//disrupt calling SystemFlowControl via MAIN() when mode is switched and call SwitchMode()
IF ((SwitchToLoading.Q OR SwitchToUnloading.Q) OR NOT bFinishedSwitchMode) AND bSetStatusOn THEN
	SwitchMode(bSwitchToLoading := bLoading,
		bFinishedSwitchMode => bFinishedSwitchMode);
END_IF;

//pumps
PU305.GetState_Profibus();
PU305(bSetStatusOnAutomatic := bSetStatusOn_PU305,
	fSetPointAutomatic := fSetPoint,
	bAlgorithmPermission := bAlgorithmPermission,
	nControlModeAutomatic := 0);
PU305.SetState_Profibus();

PU306.GetState_Profibus();
PU306(bSetStatusOnAutomatic := bSetStatusOn_PU306,
	fSetPointAutomatic := fSetPoint,
	bAlgorithmPermission := bAlgorithmPermission,
	nControlModeAutomatic := 0);
PU306.SetState_Profibus();

//valves
SV305.GetState_AI();
SV305(bSetStatusOnAutomatic := bSetStatusOn_SV305,
	fSetPointAutomatic := fSetPoint_SV305,
	bAlgorithmPermission := bAlgorithmPermission,
	nControlModeAutomatic := 0);
SV305.SetState_AO();

SV306.GetState_AI();
SV306(bSetStatusOnAutomatic := bSetStatusOn_SV306,
	fSetPointAutomatic := fSetPoint_SV306,
	bAlgorithmPermission := bAlgorithmPermission,
	nControlModeAutomatic := 0);
SV306.SetState_AO();

WMZ305(aHeatCounterTelegramm := aTelegramm_WMZ305);

IF bLoading THEN
	localState.fHeatFlowRate := -PU305.fVolumeFlowRate/3.6*4.2*(WMZ305.fFeedTemperature-WMZ305.fReturnTemperature);
	nControlMode_SV307 := 2; //cooling
ELSE
	localState.fHeatFlowRate := PU306.fVolumeFlowRate/3.6*4.2*(WMZ305.fFeedTemperature-WMZ305.fReturnTemperature);
	nControlMode_SV307 := 1; //heating
END_IF

SV307.GetState_AI();
SV307(bSetStatusOnAutomatic := bSetStatusOn_SV307,
	fSetPointAutomatic := fTemperatureBufferStorageSetPoint,
	bAlgorithmPermission := bAlgorithmPermission,
	fTemperatureExternal := fTemperatureBufferStorage,
	fThermalPowerExternal := localState.fHeatFlowRate,
	nControlModeAutomatic := nControlMode_SV307);
SV307.SetState_AO();

METHOD PROTECTED  CheckError : BOOL
VAR_INPUT
END_VAR
VAR_OUTPUT
	bError : BOOL;
END_VAR
VAR
	bError_PUx05 : BOOL;
END_VAR
//check for pump error
bError_PUx05 := PU305.bError OR PU306.bError;
END_METHOD

METHOD PROTECTED  Operational : BOOL
VAR_INPUT
END_VAR
VAR_OUTPUT
	bSwitchToWorking : BOOL := FALSE;
END_VAR
IF PU305.bStatusOn OR PU306.bStatusOn THEN
	bSwitchToWorking := TRUE;
END_IF
END_METHOD

METHOD PROTECTED  RampDown : BOOL
VAR_INPUT
END_VAR
VAR_OUTPUT
	bRampDownFinished : BOOL := FALSE;
END_VAR
bSetStatusOn_PU305 := FALSE;
bSetStatusOn_PU306 := FALSE;

IF NOT PU305.bStatusOn AND NOT PU306.bStatusOn THEN
	bSetStatusOn_SV305 := FALSE;
	bSetStatusOn_SV306 := FALSE;
	bSetStatusOn_SV307 := FALSE;
	IF SV305.fOperatingPoint<20 AND SV306.fOperatingPoint<20 AND SV307.fOperatingPoint<20 THEN
		bRampDownFinished := TRUE;
	END_IF
END_IF
END_METHOD

METHOD PROTECTED  RampUp : BOOL
VAR_INPUT
END_VAR
VAR_OUTPUT
	bRampUpFinished : BOOL := FALSE;
END_VAR
bSetStatusOn_SV305 := TRUE;
bSetStatusOn_SV306 := TRUE;
bSetStatusOn_SV307 := TRUE;

//SV307 should not be checked in ramp up to prevent chattering when sv control thermal power
IF bLoading THEN
	fSetPoint_SV305 := 100;
	fSetPoint_SV306 := 0;
	IF SV305.fOperatingPoint>80 AND SV306.fOperatingPoint<20 THEN
		bSetStatusOn_PU305 := TRUE;	
		bSetStatusOn_PU306 := FALSE;	
		bRampUpFinished := TRUE;	
	END_IF
ELSE
	fSetPoint_SV305 := 0;
	fSetPoint_SV306 := 100;
	IF SV305.fOperatingPoint<20 AND SV306.fOperatingPoint>80 THEN
		bSetStatusOn_PU305 := FALSE;	
		bSetStatusOn_PU306 := TRUE;		
		bRampUpFinished := TRUE;
	END_IF
END_IF
END_METHOD

METHOD PRIVATE SelectLocalControlMode : BOOL
VAR_INPUT
END_VAR
IF control.bManualModeActivated THEN
	bLoading := localSetParameters.bLoadingManual;
ELSIF control.bAlgorithmModeActivated AND bAlgorithmPermission THEN
	bLoading := localSetParameters.bLoadingAlgorithm;
ELSE
	bLoading := bLoadingAutomatic;
END_IF
END_METHOD

METHOD PROTECTED   SetSetPointLimits : BOOL
VAR_INPUT
END_VAR
aSetPointLimits[1] := localDefaultParameters.aSetPointLimitsTemperature[1];
aSetPointLimits[2] := localDefaultParameters.aSetPointLimitsTemperature[2];
END_METHOD

METHOD PROTECTED  SetState : BOOL
VAR_INPUT
END_VAR
VAR_OUTPUT
END_VAR
IF bLoading THEN
	fOperatingPoint := PU305.fOperatingPoint;
ELSE
	fOperatingPoint := PU306.fOperatingPoint;
END_IF

IF PU305.bStatusOn THEN
	localState.bLoading := TRUE;
ELSE
	localState.bLoading := FALSE;		
END_IF

controlState.bStatusOn := bSetStatusOn;
setPointState.aSetPointLimits := aSetPointLimits;
setPointState.fSetPoint := fSetPoint;
setPointState.fOperatingPoint := fOperatingPoint;
setPointState.sSetPointUnit := 'percent';
setPointState.sOperatingPointUnit := 'percent';
END_METHOD

PROPERTY ST_DefaultParameters : REFERENCE TO ST_VSIStorageSystemDefaultParameters
SET
localDefaultParameters := ST_DefaultParameters;
END_SET
END_PROPERTY

METHOD PRIVATE SwitchMode : BOOL
VAR_INPUT
	bSwitchToLoading : BOOL; //if false switch to cooling
END_VAR
VAR_OUTPUT
	bFinishedSwitchMode : BOOL := FALSE;
END_VAR
VAR_INST
	bRampDownFinished : BOOL := FALSE;
END_VAR
//check system state
IF bRampDownFinished THEN
	IF bSwitchToLoading THEN
		fSetPoint_SV305 := 100;
		fSetPoint_SV306 := 0;
		IF SV305.fOperatingPoint>80 AND SV306.fOperatingPoint<20 THEN
			//reset instant variable and switch on pump
			bRampDownFinished := FALSE;			
			bFinishedSwitchMode := TRUE;
			bSetStatusOn_PU305 := TRUE;
		END_IF
		
	ELSE
		fSetPoint_SV305 := 0;
		fSetPoint_SV306 := 100;
		IF SV305.fOperatingPoint<20 AND SV306.fOperatingPoint>80 THEN
			//reset instant variable and switch on pump
			bRampDownFinished := FALSE;			
			bFinishedSwitchMode := TRUE;
			bSetStatusOn_PU306 := TRUE;
		END_IF
	END_IF
ELSE
	bSetStatusOn_PU305 := FALSE;
	bSetStatusOn_PU306 := FALSE;
	IF NOT PU305.bStatusOn AND NOT PU306.bStatusOn THEN
		bRampDownFinished := TRUE;
	END_IF
END_IF
END_METHOD

METHOD PROTECTED  Working : BOOL
VAR_INPUT
END_VAR
VAR_OUTPUT
	bSwitchToOperational : BOOL := FALSE;
END_VAR
//empty method
END_METHOD

END_FUNCTION_BLOCK

// ---- POUs/03 Storages/FB_VSIStorage.TcPOU
FUNCTION_BLOCK FB_VSIStorage
VAR_INPUT
END_VAR
VAR_OUTPUT
	{attribute 'OPC.UA.DA' := '1'}	
	localState : ST_VSIStorageState;
END_VAR
VAR
	UpperTemperatureSensor : FB_TemperatureSensor; //upper temperature sensor
	MidTemperatureSensor : FB_TemperatureSensor; //mid temperature sensor
	LowerTemperatureSensor : FB_TemperatureSensor; //lower temperature sensor
END_VAR

//sensors
UpperTemperatureSensor();
MidTemperatureSensor();
LowerTemperatureSensor();

//get sensor inputs
UpperTemperatureSensor.GetState_AI();
MidTemperatureSensor.GetState_AI();
LowerTemperatureSensor.GetState_AI();

//set outputs
localState.fUpperTemperature := UpperTemperatureSensor.fTemperature;
localState.fMidTemperature := MidTemperatureSensor.fTemperature;
localState.fLowerTemperature := LowerTemperatureSensor.fTemperature;

END_FUNCTION_BLOCK

// ---- POUs/01 Actuators/ConsumerUnits/FB_MAFAC_Java.TcPOU
FUNCTION_BLOCK FB_MAFAC_Java
VAR_INPUT
END_VAR
VAR_OUTPUT
	bStatusOn : BOOL;
	bError_Connection : BOOL;
END_VAR
VAR
	OPC_UA				: FB_OPC_UA_READ;
	stOPC_UA_Server		: ST_OPC_UA_Server;
	sOPC_UA_Server_URL 	: STRING;
	sNamespaceName		: STRING;
	aNodes				: ARRAY[1..1] OF ST_OPC_UANode;
	nNodeCount			: UDINT := 1;
	stIndexRange		: ARRAY [1..nMaxIndexRange] OF ST_UAIndexRange;
	currentNode			: UDINT := 1;
	
	bStatusOn_CoolingLubricant : BOOL;
	bStatusOn_Machine : BOOL;
	
	// timer
	bStartTimer : BOOL;
	Timer : TON;
END_VAR

sOPC_UA_Server_URL 	:= GlobalVariables.sIP_MAFAC_Java;
sNamespaceName 		:= 'http://www.boschrexroth.com/IndraLogic';

(*Define Nodes to Read*)
aNodes[1].NodeID.sIdentifier			:= 'Application.UserVarGlobal.Beheizung_rot_Aktiv';
aNodes[1].NodeID.eIdentifierType		:= eUAIdentifierType_String;
aNodes[1].SizeOfDataType				:= SIZEOF(eUAType_Boolean);
aNodes[1].NodeAddInfo.nIndexRangeCount 	:= 0;
aNodes[1].NodeAddInfo.stIndexRange		:= stIndexRange;
aNodes[1].TargetVar						:= ADR(bStatusOn);
bError_Connection := OPC_UA.bError_Connection;
Timer(IN := bStartTimer,
	PT := T#5S);

bStartTimer := TRUE;
IF Timer.Q THEN
	OPC_UA(
		stNode				:= aNodes[currentNode],
		sOPC_UA_Server_Url 	:= sOPC_UA_Server_URL,
		sNamespaceName		:= sNamespaceName);
	currentNode := currentNode + 1;
	IF currentNode > nNodeCount THEN
		currentNode := 1;
	END_IF
	bStartTimer := FALSE;
END_IF

END_FUNCTION_BLOCK

// ---- POUs/01 Actuators/ConsumerUnits/FB_BvL_CleaningSystem.TcPOU
FUNCTION_BLOCK FB_BvL_CleaningSystem
VAR_INPUT
END_VAR
VAR_OUTPUT
	bError_Connection : BOOL;
	bHNHT_Demand : BOOL; 
END_VAR
VAR
	//I/O-Links
	Technical_Heat_RZ_SV AT %I* : BOOL;
	Technical_Heat_RZ_PWW AT %I* : BOOL;
	Technical_Heat_RZ_UWP AT %I* : BOOL;
	Technical_Heat_SZ_SV AT %I* : BOOL;
	Technical_Heat_SZ_PWW AT %I* : BOOL;
	Technical_Heat_SZ_UWP AT %I* : BOOL; 
	ConnectionStatus_OPC_BvL AT %I* : BOOL;
END_VAR

bHNHT_Demand := (Technical_Heat_RZ_PWW OR Technical_Heat_RZ_SV OR Technical_Heat_RZ_UWP OR Technical_Heat_SZ_PWW OR Technical_Heat_SZ_SV OR Technical_Heat_SZ_UWP) AND ConnectionStatus_OPC_BvL;
bError_Connection := NOT ConnectionStatus_OPC_BvL;

END_FUNCTION_BLOCK

// ---- POUs/05 Thermal Networks/FB_Ambient.TcPOU
FUNCTION_BLOCK FB_Ambient
VAR_INPUT
	sIPAddress : STRING(15);
END_VAR
VAR_OUTPUT
	{attribute 'OPC.UA.DA' := '1'}
	localState : ST_AmbientState;
END_VAR
VAR
	WeatherStation : FB_WeatherStation;
	AmbientTemperatureSensor_Container : FB_TemperatureSensor_KL3214;
	HallTemperatureSensor_Section1 : FB_TemperatureSensor;
	HallTemperatureSensor_Section2 : FB_TemperatureSensor;
	HallTemperatureSensor_Section3 : FB_TemperatureSensor;
	RoomTemperatureSensor_Container : FB_TemperatureSensor;
	
	//modbus tcp communication
	ModbusReader_250 : FB_MBReadRegs; //read regs from 250 on
	
	//define array to store data from every ModbusReader
	aModbus_250 : ARRAY [0..31] OF WORD;
	
	//modbus timer
	bReadModbus	: BOOL := FALSE;
	bWriteModbus_SeminarRoom : BOOL := FALSE; 
	bStartTimer : BOOL;
	TimerReader : TON; 
END_VAR

WeatherStation();
HallTemperatureSensor_Section1();
HallTemperatureSensor_Section1.GetState_AI();
HallTemperatureSensor_Section2();
HallTemperatureSensor_Section2.GetState_AI();
HallTemperatureSensor_Section3();
HallTemperatureSensor_Section3.GetState_AI();
AmbientTemperatureSensor_Container();
AmbientTemperatureSensor_Container.GetState_AI();
RoomTemperatureSensor_Container();
RoomTemperatureSensor_Container.GetState_AI();


//add ambient temperature rain etc. from weather station
localState.fOutsideTemperature_Container := AmbientTemperatureSensor_Container.fTemperature;
localState.fOutsideTemperature := WeatherStation.fTemperature;
localState.fOutsideTemperature_Mean := WeatherStation.fMeanTemperature;
localState.bRain := WeatherStation.bRain;
localState.fDawn := WeatherStation.fDawn;
localState.fWindSpeed := WeatherStation.fWindSpeed;
localState.fHallTemperature := HallTemperatureSensor_Section2.fTemperature;
localState.fRoomTemperature_Container := RoomTemperatureSensor_Container.fTemperature;


//Start and check timer for 2s interval
TimerReader(IN := bStartTimer,
	PT := T#2S);
	
bStartTimer := TRUE;
IF TimerReader.Q THEN
	bReadModbus := TRUE;
	bStartTimer := FALSE;	
END_IF
	

ModbusReader_250(
	sIPAddr := sIPAddress,
	nTCPPort := 502,
	nUnitID := 255,
	nQuantity := 30,
	nMBAddr := 250,
	cbLength := 60,
	pDestAddr := ADR(aModbus_250),
	bExecute := bReadModbus,
	tTimeout  := T#20S);
	
bReadModbus := FALSE;

//seminar room
localState.fTemperatureSeminarRoom := INT_TO_REAL(WORD_TO_INT(aModbus_250[19]))/10; 
localState.fCO2SeminarRoom := INT_TO_REAL(WORD_TO_INT(aModbus_250[17])); 
//student room
localState.fTemperatureStudentRoom := INT_TO_REAL(WORD_TO_INT(aModbus_250[28])); 
localState.fCO2StudentRoom := INT_TO_REAL(WORD_TO_INT(aModbus_250[27]));

METHOD GetState : BOOL
VAR_INPUT
END_VAR
//seminar room
localState.fTemperatureSeminarRoom := INT_TO_REAL(WORD_TO_INT(aModbus_250[19]))/10; 
localState.fCO2SeminarRoom := INT_TO_REAL(WORD_TO_INT(aModbus_250[17])); 

//student room
localState.fTemperatureStudentRoom := INT_TO_REAL(WORD_TO_INT(aModbus_250[28])); 
localState.fCO2StudentRoom := INT_TO_REAL(WORD_TO_INT(aModbus_250[27]));
END_METHOD

END_FUNCTION_BLOCK

// ---- POUs/02 Sensors/FB_WeatherStation.TcPOU
FUNCTION_BLOCK FB_WeatherStation
VAR_INPUT
END_VAR
VAR_OUTPUT
	fWindSpeed 		: REAL;
	fTemperature	: REAL;
	fMeanTemperature : REAL;
	fDawn 			: REAL;
	bRain 			: BOOL;
END_VAR
VAR
	bInit_done : BOOL := FALSE;
	
	// communication with KL6301 terminal
	KL6301_Terminal			: KL6301;
	KL6301_Error_Trigger	: r_Trig;
	KL6301_group_0_0_1		: EIB_GROUP_ADDR := (MAIN:=0, SUB_MAIN:=0, NUMBER:=1);
	KL6301_IN 				AT %I* : ARRAY[1..24]OF BYTE;
	KL6301_OUT 				AT %Q* : ARRAY[1..24]OF BYTE;
	
	Group_0_0_1		: EIB_GROUP_ADDR := (MAIN:=0,SUB_MAIN:=0,NUMBER:=1);
	Group_0_0_2		: EIB_GROUP_ADDR := (MAIN:=0,SUB_MAIN:=0,NUMBER:=2);
	Group_0_0_3		: EIB_GROUP_ADDR := (MAIN:=0,SUB_MAIN:=0,NUMBER:=3);
	Group_0_0_4		: EIB_GROUP_ADDR := (MAIN:=0,SUB_MAIN:=0,NUMBER:=4);

	recWindSpeed	: EIB_2OCTET_FLOAT_REC;
	recTemperature	: EIB_2OCTET_FLOAT_REC;
	recDawn			: EIB_2OCTET_FLOAT_REC;
	recRain			: EIB_BIT_REC;
	
	//clock
	stDefaultParameters_Clock : ST_ClockDefaultParameters := (tTaskCycleTime := GlobalVariables.tCtrlCycleTime_MAIN, tCtrlCycleTime := T#1M);
	Clock : FB_Clock := (ST_DefaultParameters := stDefaultParameters_Clock);
	Moving_Average_Temperature : FB_CTRL_MOVING_AVERAGE;
	bInit_Average_Temperature : BOOL;
END_VAR

//initialize clock
Clock();

//read and write to terminal
KL6301_Terminal(KL6301_IN:=KL6301_IN, KL6301_OUT:=KL6301_OUT);
KL6301_Error_Trigger(CLK := KL6301_Terminal.bError);

//initialize terminal
IF (NOT bInit_done) THEN
	bInit_done := InitializeTerminal();
END_IF

IF(KL6301_Terminal.bReady) THEN
	recWindSpeed(
		Group_Address := Group_0_0_1,
		strData_Rec := KL6301_Terminal.str_Data_Rec
	);

	recTemperature(
		Group_Address := Group_0_0_2,
		strData_Rec := KL6301_Terminal.str_Data_Rec
	);

	recDawn(
		Group_Address := Group_0_0_3,
		strData_Rec := KL6301_Terminal.str_Data_Rec
	);

	recRain(
		Group_Address := Group_0_0_4,
		strData_Rec := KL6301_Terminal.str_Data_Rec
	);

	fWindSpeed := recWindSpeed.rData;
	fTemperature := recTemperature.rData;
	fDawn := recDawn.rData;
	bRain := recRain.bData;
END_IF

//calculate moving average temperatrue
CalculateAverageTemperature(fActualTemperature := fTemperature, fMeanTemperature => fMeanTemperature);

METHOD CalculateAverageTemperature : REAL
VAR_INPUT
	fActualTemperature : REAL;
END_VAR
VAR_OUTPUT
	fMeanTemperature : REAL;
END_VAR
VAR_INST
	fTemperature_init : REAL;
	fHours_Moving_Average : UINT := 6;
	fMeanTemperature_Summer_init : REAL := 22;
	fMeanTemperature_Winter_init : REAL := 5;
	
	stParameters_Average_Temperature : ST_CTRL_MOVING_AVERAGE_PARAMS;
	aTemperatureBuffer 				: ARRAY [1..360] OF FLOAT := [360(15)];
END_VAR
//calculate initialization temperature
IF Clock.stClockState.sintMonth>4 AND Clock.stClockState.sintMonth<10 THEN
	//summer
	fTemperature_init := fMeanTemperature_Summer_init;
ELSE
	//winter	
	fTemperature_init := fMeanTemperature_Winter_init;
END_IF

stParameters_Average_Temperature.tCtrlCycleTime := T#60S;
stParameters_Average_Temperature.tTaskCycleTime := GlobalVariables.tTaskCycleTime_MAIN;
stParameters_Average_Temperature.nSamplesToFilter := fHours_Moving_Average*60; (* 1min= 60 sec*)
stParameters_Average_Temperature.pWorkArray_ADR := ADR(aTemperatureBuffer);
stParameters_Average_Temperature.nWorkArray_SIZEOF := SIZEOF(aTemperatureBuffer);

Moving_Average_Temperature(
	fIn := fActualTemperature,
	fManSyncValue := 15,
	bSync := FALSE,
	eMode := 2,
	bHold := FALSE,
	stParams := stParameters_Average_Temperature);
fMeanTemperature := LREAL_TO_REAL(Moving_Average_Temperature.fOut);
END_METHOD

METHOD InitializeTerminal : BOOL
VAR_INPUT
END_VAR
VAR_OUTPUT
	bInit_done : BOOL := FALSE;
END_VAR
KL6301_Terminal.EIB_PHYS_ADDR.Area:=1;
KL6301_Terminal.EIB_PHYS_ADDR.Line:=1;
KL6301_Terminal.EIB_PHYS_ADDR.Device:=5;
KL6301_Terminal.EIB_GROUP_FILTER[1].GROUP_ADDR:=KL6301_group_0_0_1;
KL6301_Terminal.EIB_GROUP_FILTER[1].GROUP_LEN:=12;
KL6301_Terminal.idx:=1;
KL6301_Terminal.iMode:=1;

IF(KL6301_Terminal.bReady) THEN
	bInit_done := TRUE;
END_IF

IF KL6301_Error_Trigger.Q THEN
	KL6301_Terminal.bActivate:=FALSE;
ELSE
	KL6301_Terminal.bActivate:=TRUE;
END_IF
END_METHOD

METHOD ReadValues : BOOL
VAR_INPUT
END_VAR
VAR_OUTPUT
	fWindSpeed 		: REAL;
	fTemperature	: REAL;
	fDawn 			: REAL;
	bRain 			: BOOL;
END_VAR
VAR

END_VAR
END_METHOD

END_FUNCTION_BLOCK

// ---- POUs/02 Sensors/FB_LowVoltageMainDistribution.TcPOU
FUNCTION_BLOCK FB_LowVoltageMainDistribution
VAR_INPUT
END_VAR
VAR_OUTPUT
END_VAR
VAR
	EM_Offices : FB_ElectricityMeter_ABBA44113100;
	EM_ProductionHall_HVAC : FB_ElectricityMeter_ABBA44113100;
	EM_ProductionHall_Lighting : FB_ElectricityMeter_ABBA44113100;
	EM_TotalBuilding : FB_ElectricityMeter_ABBA44213100;
END_VAR

EM_Offices(aElectricityMeterTelegramm := Telegramm_SZ_Buerotrakt);
EM_ProductionHall_HVAC(aElectricityMeterTelegramm := Telegramm_SZ_Halle_TGA);
EM_ProductionHall_Lighting(aElectricityMeterTelegramm := Telegramm_SZ_Halle_Licht);
EM_TotalBuilding(aElectricityMeterTelegramm := Telegramm_SZ_Gebaeude);

END_FUNCTION_BLOCK

// ---- POUs/01 Actuators/ConsumerUnits/FB_Ventilation.TcPOU
FUNCTION_BLOCK FB_Ventilation EXTENDS FB_ActuatorContinous
VAR_INPUT
	sIPAddress : STRING(15);
	 //default value 
	bSetStatusOn_SeminarRoom : BOOL:= FALSE;
	bSetStatusOn_Hall : BOOL := FALSE; 
	bSetStatusOn_HiwiRoom : BOOL := FALSE; 
	bSetStatusOn_ClimateRoom : BOOL := FALSE;
	risingEdge_Trigger : R_TRIG; 
	fallingEdge_Trigger : F_TRIG; 
	bExecute_ClimateRoom : BOOL := FALSE; 
	
END_VAR
VAR_OUTPUT
	fReturnTemperature : REAL;
	bError : BOOL;
END_VAR
VAR
	
	{attribute 'OPC.UA.DA' := '1'}
	localState : ST_VentilationState;
	
	//default parameters
	localDefaultParameters : ST_VentilationDefaultParameters;	
	

	//modbus tcp communication
	ModbusReader_100 : FB_MBReadRegs; //read regs from 100 on
	ModbusReader_135 : FB_MBReadInputs; 
	ModbusReader_112 : FB_MBReadInputs; 
	ModbusReader_166 : FB_MBReadInputs; 
	ModbusReader_167 : FB_MBReadInputs; 
	ModbusReader_168 : FB_MBReadInputs;
	ModbusReader_169 : FB_MBReadInputs;  
	ModbusReader_200 : FB_MBReadRegs; 
	
	
	ModbusWrite_100 : FB_MBWriteSingleCoil; // write reg 100
	ModbusWrite_101 : FB_MBWriteSingleCoil; // write reg 101
	ModbusWrite_102 : FB_MBWriteSingleCoil; // Write reg 102
	ModbusWrite_103 : FB_MBWriteSingleCoil; // Write reg 103
	ModbusWrite_203 : FB_MBWriteSingleCoil; // Write reg 203
	ModbusWrite_213 : FB_MBWriteSingleCoil; // Write reg 213
	
	
	
	//define array to store data from every ModbusReader
	aModbus_100 : ARRAY [0..14] OF WORD;
	aModbus_112 : ARRAY [0..0] OF BYTE;
	aModbus_135 : ARRAY [0..3] OF BYTE;
	aModbus_166 : ARRAY [0..0] OF BYTE;
	aModbus_167 : ARRAY [0..0] OF BYTE;
	aModbus_168 : ARRAY [0..0] OF BYTE;
	aModbus_169 : ARRAY [0..0] OF BYTE;
	aModbus_200 : ARRAY [0..50] OF WORD;

	
	//modbus timer
	bReadModbus	: BOOL := FALSE;
	
	//write SeminarRoom
	bWriteModbus_SeminarRoom : BOOL := FALSE; 
	bSendValue_SeminarRoom : BOOL := FALSE; 
	iStep_SeminarRoom : INT := 0;
	
	//write Productionhall
	bWriteModbus_Hall : BOOL := FALSE;
	bSendValue_Hall :BOOL := FALSE;
	iStep_Hall : INT := 0; // 0 = IDLE, 1 = Write FALSE vlaue to modbus, 2 = Wait after sending FALSE
	
	//write Studentroom
	bWriteModbus_StudentRoom : BOOL := FALSE; 
	bSendValue_StudentRoom : BOOL := FALSE;
	iStep_StudentRoom : INT := 0; 
	
	//write ClimateRoom
	bWriteModbus_ClimateRoom : BOOL := FALSE;
	bSendValue_ClimateRoom :BOOL := FALSE;
	iStep_ClimateRoom : INT := 0; // 0 = IDLE, 1 = Write FALSE vlaue to modbus, 2 = Wait after sending FALSE
	
	

	bStartTimer : BOOL;
	TimerReader : TON;
	TimerSeminarRoom : TON; 
	TimerHall : TON;
	TimerStudentRoom : TON; 
	TimerClimateRoom : TON;  
	bStartTimerSeminarRoom : BOOL; 
	bStartTimerHall : BOOL; 
	bStartTimerStudentRoom : BOOL; 
	bStartTimerClimateRoom : BOOL; 
	
	//read single status 
	bStatusSeminarRoom : BOOL; 
	bStatusProductionHall : BOOL; 
	bStatusHiwiRoom : BOOL; 
	bStatusClimateRoom : BOOL; 
	
END_VAR


//Start and check timer for 2s interval
TimerReader(IN := bStartTimer, PT := T#1S);

bStartTimer := TRUE;
IF TimerReader.Q THEN
    bReadModbus := TRUE;      
    bStartTimer := FALSE;  
END_IF

(*ModbusReader_100(
	sIPAddr := sIPAddress,
	nTCPPort := 502,
	nUnitID := 255,
	nQuantity := 8,
	nMBAddr := 100,
	cbLength := 16,
	pDestAddr := ADR(aModbus_100),
	bExecute := bReadModbus,
	tTimeout  := T#20S);*)

// read status experiment mode
ModbusReader_112(
	sIPAddr := sIPAddress,
	nTCPPort := 502,
	nUnitID := 1,
	nQuantity := 1,
	nMBAddr := 112,
	cbLength := 1,
	pDestAddr := ADR(aModbus_112),
	bExecute := bReadModbus,
	tTimeout  := T#20S);

bReadModbus := bReadModbus AND NOT ModbusReader_135.bBusy;
	
ModbusReader_135(
	sIPAddr := sIPAddress,
	nTCPPort := 502,
	nUnitID := 16#FF,
	nQuantity := 4,
	nMBAddr := 166,
	cbLength := SIZEOF(aModbus_135),
	pDestAddr := ADR(aModbus_135),
	bExecute := bReadModbus,
	tTimeout  := T#20S);

//unpack the four bits in 166 in bool values
bStatusSeminarRoom := (aModbus_135[0] AND 16#01) <> 0; // Input 166
bStatusProductionHall := (aModbus_135[0] AND 16#02) <> 0; // Input 167
bStatusHiwiRoom := (aModbus_135[0] AND 16#04) <> 0; // Input 168
bStatusClimateRoom := (aModbus_135[0] AND 16#08) <> 0; // Input 169

localState.bStatusOnSeminarRoom := bStatusSeminarRoom;
localState.bStatusOnProductionHall := bStatusProductionHall; 
localState.bStatusOnStudentRoom := bStatusHiwiRoom; 
localState.bStatusOnClimateRoom := bStatusClimateRoom; 

(*ModbusReader_200(
	sIPAddr := sIPAddress,
	nTCPPort := 502,
	nUnitID := 255,
	nQuantity := 49,
	nMBAddr := 135,
	cbLength := 98,
	pDestAddr := ADR(aModbus_200),
	bExecute := bReadModbus,
	tTimeout  := T#20S);*)

	
bReadModbus := FALSE;

METHOD GetState : BOOL
VAR_INPUT
END_VAR
//empty method (abstract method)
END_METHOD

METHOD PROTECTED SelectSetPoint : BOOL
VAR_INPUT
END_VAR
IF control.bManualModeActivated THEN
	fsetPoint := setSetPoint.fSetPointManual;
ELSIF control.bAlgorithmModeActivated AND bAlgorithmPermission THEN
	fsetPoint := setSetPoint.fSetPointAlgorithm;
ELSE
	fsetPoint := fSetPointAutomatic;
END_IF
END_METHOD

METHOD PROTECTED  SetSetPointLimits : BOOL
VAR_INPUT
END_VAR
aSetPointLimits[1] := localDefaultParameters.aSetPointLimitsTemperature[1];
aSetPointLimits[2] := localDefaultParameters.aSetPointLimitsTemperature[2];
END_METHOD

METHOD SetState : BOOL
VAR_INPUT
END_VAR
TimerSeminarRoom(IN := bStartTimerSeminarRoom,
	PT := T#500MS);
	
TimerHall(IN := bStartTimerHall,
	PT := T#500MS);
	
TimerStudentRoom(IN := bStartTimerStudentRoom,
	PT := T#500MS);

TimerClimateRoom(IN := bStartTimerClimateRoom,
	PT := T#500MS);
	

	
CASE iStep_SeminarRoom OF
	0: // check for change in status
		IF (bSetStatusOn_SeminarRoom = TRUE AND localstate.bStatusOnSeminarRoom= FALSE) OR (bSetStatusOn_SeminarRoom = FALSE AND localState.bStatusOnSeminarRoom = TRUE) THEN
			bWriteModbus_SeminarRoom := TRUE;
			bSendValue_SeminarRoom := TRUE;
			bStartTimerSeminarRoom := TRUE;
			iStep_SeminarRoom := 1; 
			// go to next step
		END_IF 
	1: // wait for timer to end then write FALSE
		IF TimerSeminarRoom.Q THEN
			bWriteModbus_SeminarRoom := TRUE;
			bSendValue_SeminarRoom := FALSE;
			bStartTimerSeminarRoom := FALSE;
			iStep_SeminarRoom := 2;	
		END_IF
	2: // time for waiting before check starts again
		bStartTimerSeminarRoom := TRUE;
		IF TimerSeminarRoom.Q THEN
			iStep_SeminarRoom := 0;
		END_IF
		
END_CASE

ModbusWrite_100(
	sIPAddr := sIPAddress, 
	nTCPPort := 502, 
	nUnitID := 16#FF, 
	nMBAddr := 100, 
	nValue := SEL(bSendValue_SeminarRoom, WORD#16#0000, WORD#16#FF00),
	bExecute := bWriteModbus_SeminarRoom, 
	tTimeout := T#20S);

bWriteModbus_SeminarRoom := FALSE; 



CASE iStep_Hall OF
	0: // check for change in status
		IF (bSetStatusOn_Hall = TRUE AND localstate.bStatusOnProductionHall= FALSE) OR (bSetStatusOn_Hall = FALSE AND localState.bStatusOnProductionHall = TRUE) THEN
			bWriteModbus_Hall := TRUE;
			bSendValue_Hall := TRUE;
			bStartTimerHall := TRUE;
			iStep_Hall := 1; 
			// go to next step
		END_IF 
	1: // wait for timer to end then write FALSE
		IF TimerHall.Q THEN
			bWriteModbus_Hall := TRUE;
			bSendValue_Hall := FALSE;
			bStartTimerHall := FALSE;
			iStep_Hall := 2;	
		END_IF
	2: // time for waiting before check starts again
		bStartTimerHall := TRUE;
		IF TimerHall.Q THEN
			iStep_Hall := 0;
		END_IF
		
END_CASE

ModbusWrite_101(
	sIPAddr := sIPAddress, 
	nTCPPort := 502, 
	nUnitID := 16#FF, 
	nMBAddr := 101, 
	nValue := SEL(bSendValue_Hall, WORD#16#0000, WORD#16#FF00),
	bExecute := bWriteModbus_Hall, 
	tTimeout := T#20S); 
	
bWriteModbus_Hall := FALSE; 

	
CASE iStep_StudentRoom OF
	0: // check for change in status
		IF (bSetStatusOn_HiwiRoom = TRUE AND localstate.bStatusOnStudentRoom= FALSE) OR (bSetStatusOn_HiwiRoom = FALSE AND localState.bStatusOnStudentRoom = TRUE) THEN
			bWriteModbus_StudentRoom := TRUE;
			bSendValue_StudentRoom := TRUE;
			bStartTimerStudentRoom := TRUE;
			iStep_StudentRoom := 1; 
			// go to next step
		END_IF 
	1: // wait for timer to end then write FALSE
		IF TimerStudentRoom.Q THEN
			bWriteModbus_StudentRoom := TRUE;
			bSendValue_StudentRoom := FALSE;
			bStartTimerStudentRoom := FALSE;
			iStep_StudentRoom := 2;	
		END_IF
	2: // time for waiting before check starts again
		bStartTimerStudentRoom := TRUE;
		IF TimerStudentRoom.Q THEN
			iStep_StudentRoom := 0;
		END_IF
		
END_CASE

ModbusWrite_102(
	sIPAddr := sIPAddress, 
	nTCPPort := 502, 
	nUnitID := 16#FF, 
	nMBAddr := 107, 
	nValue := SEL(bSendValue_StudentRoom, WORD#16#0000, WORD#16#FF00),
	bExecute := bWriteModbus_StudentRoom, 
	tTimeout := T#20S); 
	
bWriteModbus_StudentRoom := FALSE;  
	
	
CASE iStep_ClimateRoom OF
	0: // check for change in status
		IF (bSetStatusOn_ClimateRoom = TRUE AND localstate.bStatusOnClimateRoom = FALSE) OR (bSetStatusOn_ClimateRoom = FALSE AND localState.bStatusOnClimateRoom = TRUE) THEN
			bWriteModbus_ClimateRoom := TRUE;
			bSendValue_ClimateRoom := TRUE;
			bStartTimerClimateRoom := TRUE;
			iStep_ClimateRoom := 1; 
			// go to next step
		END_IF 
	1: // wait for timer to end then write FALSE
		IF TimerClimateRoom.Q THEN
			bWriteModbus_ClimateRoom := TRUE;
			bSendValue_ClimateRoom := FALSE;
			bStartTimerClimateRoom := FALSE;
			iStep_ClimateRoom := 2;	
		END_IF
	2: // time for waiting before check starts again
		bStartTimerClimateRoom := TRUE;
		IF TimerClimateRoom.Q THEN
			iStep_ClimateRoom := 0;
		END_IF
		
END_CASE

ModbusWrite_103(
	sIPAddr := sIPAddress, 
	nTCPPort := 502, 
	nUnitID := 16#FF, 
	nMBAddr := 108, 
	nValue := SEL(bSendValue_ClimateRoom, WORD#16#0000, WORD#16#FF00),
	bExecute := bWriteModbus_ClimateRoom,
	tTimeout := T#20S);

bWriteModbus_ClimateRoom := FALSE;
END_METHOD

END_FUNCTION_BLOCK

// ---- POUs/04 Systems/CoolingSystems/FB_AbsorptionChillerSystem.TcPOU
FUNCTION_BLOCK FB_AbsorptionChillerSystem EXTENDS FB_SystemContinous
VAR_INPUT
END_VAR
VAR_OUTPUT
END_VAR
VAR
	//default parameters
	localDefaultParameters : ST_AbsorptionChillerDefaultParameters;

	//pumps
	stPU341DefaultParameters : ST_PumpGrundfosMagna3DefaultParameters := (bPumpBeforeApplication := TRUE, tTaskCycleTime := GlobalVariables.tTaskCycleTime_MAIN, tCtrlCycleTime := GlobalVariables.tCtrlCycleTime_MAIN);
	stPU241DefaultParameters : ST_PumpGrundfosMagna3DefaultParameters := (bPumpBeforeApplication := FALSE, tTaskCycleTime := GlobalVariables.tTaskCycleTime_MAIN, tCtrlCycleTime := GlobalVariables.tCtrlCycleTime_MAIN);
	stPU141DefaultParameters : ST_PumpGrundfosMagna3DefaultParameters := (bPumpBeforeApplication := FALSE, tTaskCycleTime := GlobalVariables.tTaskCycleTime_MAIN, tCtrlCycleTime := GlobalVariables.tCtrlCycleTime_MAIN);
	PU341 : FB_PumpGrundfosMagna3 := (ST_DefaultParameters := stPU341DefaultParameters);
	PU241 : FB_PumpGrundfosMagna3 := (ST_DefaultParameters := stPU241DefaultParameters);
	PU141 : FB_PumpGrundfosMagna3 := (ST_DefaultParameters := stPU141DefaultParameters);

	//valves
	stRV341DefaultParameters : ST_MixingValveDefaultParameters := (bFeedbackSignal := FALSE, tTaskCycleTime := GlobalVariables.tCtrlCycleTime_MAIN, tCtrlCycleTime := GlobalVariables.tCtrlCycleTime_MAIN);
	stRV241DefaultParameters : ST_MixingValveDefaultParameters := (bFeedbackSignal := FALSE, tTaskCycleTime := GlobalVariables.tCtrlCycleTime_MAIN, tCtrlCycleTime := GlobalVariables.tCtrlCycleTime_MAIN);
	stRV141DefaultParameters : ST_MixingValveDefaultParameters := (bFeedbackSignal := FALSE, tTaskCycleTime := GlobalVariables.tCtrlCycleTime_MAIN, tCtrlCycleTime := GlobalVariables.tCtrlCycleTime_MAIN);
	RV341 : FB_MixingValve := (ST_DefaultParameters := stRV341DefaultParameters);
	RV241 : FB_MixingValve := (ST_DefaultParameters := stRV241DefaultParameters);
	RV141 : FB_MixingValve := (ST_DefaultParameters := stRV141DefaultParameters);
	
	//internal variables
	bSetStatusOn_PU341 : BOOL;
	bSetStatusOn_PU241 : BOOL;
	bSetStatusOn_PU141 : BOOL;
	bSetStatusOn_RV341 : BOOL;
	bSetStatusOn_RV241 : BOOL;
	bSetStatusOn_RV141 : BOOL;
	
	//timer
	bStartTimer : BOOL;
	Timer : TON;
END_VAR

MAIN();

//pumps
PU341.GetState_Profibus();
PU341(bSetStatusOnAutomatic := bSetStatusOn_PU341,
	fSetPointAutomatic := 100,
	bAlgorithmPermission := bAlgorithmPermission,
	nControlModeAutomatic := 0);
PU341.SetState_Profibus();

PU241.GetState_Profibus();
PU241(bSetStatusOnAutomatic := bSetStatusOn_PU241,
	fSetPointAutomatic := 100,
	bAlgorithmPermission := bAlgorithmPermission,
	nControlModeAutomatic := 0);
PU241.SetState_Profibus();

PU141.GetState_Profibus();
PU141(bSetStatusOnAutomatic := bSetStatusOn_PU141,
	fSetPointAutomatic := 100,
	bAlgorithmPermission := bAlgorithmPermission,
	nControlModeAutomatic := 0);
PU141.SetState_Profibus();

//use timer because valve has no feedback signal (75 sec)
Timer(IN := bStartTimer,
	PT := T#75S);

//valves
RV341.GetState_AI();
RV341(bSetStatusOnAutomatic := bSetStatusOn_RV341,
	fSetPointAutomatic := fSetPoint,
	bAlgorithmPermission := bAlgorithmPermission,
	fTemperatureExternal := PU341.fTemperatureInternal,
	nControlModeAutomatic := 0);
RV341.SetState_AO();

RV341.GetState_AI();
RV341(bSetStatusOnAutomatic := bSetStatusOn_RV341,
	fSetPointAutomatic := 85,
	bAlgorithmPermission := bAlgorithmPermission,
	fTemperatureExternal := PU341.fTemperatureInternal,
	nControlModeAutomatic := 1);
RV341.SetState_AO();

RV241.GetState_AI();
RV241(bSetStatusOnAutomatic := bSetStatusOn_RV241,
	fSetPointAutomatic := 32,
	bAlgorithmPermission := bAlgorithmPermission,
	fTemperatureExternal := PU241.fTemperatureExternal,
	nControlModeAutomatic := 2);
RV241.SetState_AO();

RV141.GetState_AI();
RV141(bSetStatusOnAutomatic := bSetStatusOn_RV241,
	fSetPointAutomatic := fSetPoint,
	bAlgorithmPermission := bAlgorithmPermission,
	fTemperatureExternal := PU241.fTemperatureInternal,
	nControlModeAutomatic := 1);
RV141.SetState_AO();

METHOD PROTECTED  CheckError : BOOL
VAR_INPUT
END_VAR
VAR_OUTPUT
	bError : BOOL;
END_VAR
bError := PU341.bError OR PU241.bError OR PU141.bError;
END_METHOD

METHOD PROTECTED  Operational : BOOL
VAR_INPUT
END_VAR
VAR_OUTPUT
	bSwitchToWorking : BOOL := FALSE;
END_VAR
bSetStatusOn_PU341 := TRUE;
bSetStatusOn_PU241 := TRUE;
bSetStatusOn_PU141 := TRUE;

IF PU341.bStatusOn AND PU241.bStatusOn AND PU141.bStatusOn THEN
	bSwitchToWorking := TRUE;
END_IF
END_METHOD

METHOD PROTECTED  RampDown : BOOL
VAR_INPUT
END_VAR
VAR_OUTPUT
	bRampDownFinished : BOOL := FALSE;
END_VAR
bSetStatusOn_PU341 := FALSE;
bSetStatusOn_PU241 := FALSE;
bSetStatusOn_PU141 := FALSE;

IF NOT PU341.bStatusOn AND NOT PU241.bStatusOn AND NOT PU141.bStatusOn THEN
	bStartTimer := TRUE;
	bSetStatusOn_RV341 := FALSE;
	bSetStatusOn_RV241 := FALSE;
	bSetStatusOn_RV141 := FALSE;
	IF Timer.Q THEN
		bRampDownFinished := TRUE;
		bStartTimer := FALSE;
	END_IF
END_IF
END_METHOD

METHOD PROTECTED  RampUp : BOOL
VAR_INPUT
END_VAR
VAR_OUTPUT
	bRampUpFinished : BOOL := FALSE;
END_VAR
bSetStatusOn_RV341 := TRUE;
bSetStatusOn_RV241 := TRUE;
bSetStatusOn_RV141 := TRUE;
bStartTimer := TRUE;

IF Timer.Q THEN
	bRampUpFinished := TRUE;
	bStartTimer := FALSE;
END_IF
END_METHOD

METHOD PROTECTED   SetSetPointLimits : BOOL
VAR_INPUT
END_VAR
aSetPointLimits[1] := localDefaultParameters.aSetPointLimitsTemperature[1];
aSetPointLimits[2] := localDefaultParameters.aSetPointLimitsTemperature[2];
END_METHOD

METHOD PROTECTED  SetState : BOOL
VAR_INPUT
END_VAR
VAR_OUTPUT
END_VAR
fOperatingPoint := PU341.fTemperatureInternal;

controlState.bStatusOn := bSetStatusOn;
setPointState.aSetPointLimits := aSetPointLimits;
setPointState.fSetPoint := fSetPoint;
setPointState.fOperatingPoint := fOperatingPoint;
setPointState.sSetPointUnit := 'degreeC';
setPointState.sOperatingPointUnit := 'degreeC';
END_METHOD

METHOD PROTECTED  Working : BOOL
VAR_INPUT
END_VAR
VAR_OUTPUT
	bSwitchToOperational : BOOL := FALSE;
END_VAR
//empty method
END_METHOD

END_FUNCTION_BLOCK

// ---- POUs/06 Strategy/FB_StrategyController_noChiller.TcPOU
FUNCTION_BLOCK FB_StrategyController_noChiller
VAR_INPUT
	ambientState : ST_AmbientState;
	
	//actual temperatures in thermal networks
	cnState : ST_ThermalNetworkState;
	hnltState : ST_ThermalNetworkState;
	hnhtState : ST_ThermalNetworkState;
END_VAR
VAR_OUTPUT	
	cnControl : ST_CoolingNetworkControl;
	hnltControl : ST_HeatingNetworkLowTemperatureControl;	
	hnhtControl : ST_HeatingNetworkHighTemperatureControl;
	hnltCnLinkageControl : ST_HnltCnLinkageControl;
	hnhtHnltLinkageControl : ST_HnhtHnltLinkageControl;
	hnhtCnLinkageControl : ST_HnhtCnLinkageControl;
END_VAR
VAR
	{attribute 'OPC.UA.DA' := '1'}
	localSetParameters : ST_StrategySetParameters;	
	{attribute 'OPC.UA.DA' := '1'}
	localState : ST_StrategyState;	

	//default parameters
	localDefaultParameters : ST_StrategyDefaultParameters;

	//internal variables
	fTargetTemperature_HNHT_Heating : REAL;
	fTargetTemperature_HNHT_Cooling : REAL;
	fTargetTemperature_HNLT_Cooling : REAL;
	fTargetTemperature_HNLT_Heating : REAL;
	fTargetTemperature_CN : REAL;
	aTemperatureLimits_HNHT : ARRAY[1..2] OF REAL;
	aTemperatureLimits_HNLT : ARRAY[1..2] OF REAL;
	aTemperatureLimits_CN : ARRAY[1..2] OF REAL;
	stHNHTCheckDefaultParameters : ST_RangeCheckDefaultParameters := (tTaskCycleTime := GlobalVariables.tCtrlCycleTime_MAIN, tCtrlCycleTime := GlobalVariables.tCtrlCycleTime_MAIN, fRestoreDifference := 5);
	HNHT_Check : FB_RangeCheck := (ST_DefaultParameters := stHNHTCheckDefaultParameters);
	stHNLTCheckDefaultParameters : ST_RangeCheckDefaultParameters := (tTaskCycleTime := GlobalVariables.tCtrlCycleTime_MAIN, tCtrlCycleTime := GlobalVariables.tCtrlCycleTime_MAIN, fRestoreDifference := 5);
	HNLT_Check : FB_RangeCheck := (ST_DefaultParameters := stHNLTCheckDefaultParameters);
	stCNCheckDefaultParameters : ST_RangeCheckDefaultParameters := (tTaskCycleTime := GlobalVariables.tCtrlCycleTime_MAIN, tCtrlCycleTime := GlobalVariables.tCtrlCycleTime_MAIN, fRestoreDifference := 2);
	CN_Check : FB_RangeCheck := (ST_DefaultParameters := stCNCheckDefaultParameters);
	
	
	//controller and variables for high temperature heating network
	fOffset_TargetTemperature_CHP1 : REAL; //not fixed, switches depending on ambient temperature -> see method: ControlHNHT
	fOffset_TargetTemperature_CHP2 : REAL; //not fixed, switches depending on ambient temperature -> see method: ControlHNHT
	Controller_CHP_Prioritization : FB_CTRL_2POINT;
	Controller_CHP_Prioritization_Parameters : ST_CTRL_2POINT_PARAMS;	
	Controller_CHP1_UpperTemperature : FB_CTRL_2POINT; //check upper temperature for turning on chp
	Controller_CHP1_LowerTemperature : FB_CTRL_2POINT; //check lower temperature for turning off chp
	Controller_CHP1_Parameters : ST_CTRL_2POINT_PARAMS;	
	Trigger_CHP1_UpperTemperature : F_TRIG;
	Trigger_CHP1_LowerTemperature : F_TRIG;
	bTrigger_CHP1 : BOOL;
	Controller_CHP2_UpperTemperature : FB_CTRL_2POINT;
	Controller_CHP2_LowerTemperature : FB_CTRL_2POINT;
	Controller_CHP2_Parameters : ST_CTRL_2POINT_PARAMS;
	Trigger_CHP2_UpperTemperature : F_TRIG;
	Trigger_CHP2_LowerTemperature : F_TRIG;
	bTrigger_CHP2 : BOOL;
	Controller_CondensingBoiler : FB_CTRL_2POINT;
	Controller_CondensingBoiler_Parameters : ST_CTRL_2POINT_PARAMS;
	Controller_VSI_Loading_Permission : FB_CTRL_2POINT;
	Controller_VSI_Loading_Permission_Parameters : ST_CTRL_2POINT_PARAMS;
	Controller_VSI_Unloading_Permission : FB_CTRL_2POINT;
	Controller_VSI_Unloading_Permission_Parameters : ST_CTRL_2POINT_PARAMS;
	Controller_Buffer_VSI_Unloading : FB_CTRL_2POINT;
	Controller_Buffer_VSI_Unloading_Parameters : ST_CTRL_2POINT_PARAMS;
	Controller_StaticHeating : FB_CTRL_2POINT;
	Controller_StaticHeating_Parameters : ST_CTRL_2POINT_PARAMS;
	
	//controllers and variables for low temperature heating network
	Controller_OuterCapillaryTubeMats : FB_CTRL_2POINT;
	Controller_OuterCapillaryTubeMats_Parameters : ST_CTRL_2POINT_PARAMS;
	Controller_OuterCapillaryTubeMats_Permission : FB_CTRL_2POINT;
	Controller_OuterCapillaryTubeMats_Permission_Parameters : ST_CTRL_2POINT_PARAMS;
	fOffset_TargetTemperature_OuterCapillaryTubeMats_Cooling : REAL := 1;	
	fOffset_OuterCapillaryTubeMats_Permission : REAL := 10;
	
	Controller_HVFA_HNLT_HVFALoadingPermission : FB_CTRL_2POINT;
	Controller_HVFA_HNLT_HVFALoadingPermission_Parameters : ST_CTRL_2POINT_PARAMS;
	Controller_HVFA_HNLT_HVFAUnloadingPermission : FB_CTRL_2POINT;
	Controller_HVFA_HNLT_HVFAUnloadingPermission_Parameters : ST_CTRL_2POINT_PARAMS;
	Controller_Buffer_HVFA_HNLT_HVFAUnloading : FB_CTRL_2POINT;
	Controller_Buffer_HVFA_HNLT_HVFAUnloading_Parameters : ST_CTRL_2POINT_PARAMS;
	Controller_Buffer_HVFA_HNLT_HVFALoading : FB_CTRL_2POINT;
	Controller_Buffer_HVFA_HNLT_HVFALoading_Parameters : ST_CTRL_2POINT_PARAMS;
	Controller_HVFA_HNLT_Recooling : FB_CTRL_2POINT;
	Controller_HVFA_HNLT_Recooling_Parameters : ST_CTRL_2POINT_PARAMS;
	fOffset_TargetTemperature_HVFA_HNLT_Heating : REAL := 1;
	fOffset_HVFA_HNLT_Recooling : REAL := 2;
		
	
	//controllers and variables for cooling network
	fOffset_TargetTemperature_eChiller : REAL := 0.5;	
	fOffset_TargetTemperature_HVFA_CN : REAL := 1;
	fOffset_TargetTemperature_HVFA_CN_Permission : REAL := 2.5;
	Controller_eChiller : FB_CTRL_2POINT;
	Controller_eChiller_Parameters : ST_CTRL_2POINT_PARAMS;	
	Controller_HVFA_CN_LoadingPermission : FB_CTRL_2POINT;
	Controller_HVFA_CN_LoadingPermission_Parameters : ST_CTRL_2POINT_PARAMS;
	Controller_HVFA_CN_UnloadingPermission : FB_CTRL_2POINT;
	Controller_HVFA_CN_UnloadingPermission_Parameters : ST_CTRL_2POINT_PARAMS;
	Controller_Buffer_HVFA_CN_Unloading : FB_CTRL_2POINT;
	Controller_Buffer_HVFA_CN_Unloading_Parameters : ST_CTRL_2POINT_PARAMS;

	//controllers and variables for hnht and hnlt linkage
	Controller_HeatExchanger1 : FB_CTRL_2POINT;
	Controller_HeatExchanger1_Parameters : ST_CTRL_2POINT_PARAMS;
	fOffset_TargetTemperature_HeatExchanger1 : REAL := 2;
	Controller_HeatPump_HNHT : FB_CTRL_2POINT;
	Controller_HeatPump_HNHT_Parameters : ST_CTRL_2POINT_PARAMS;
	fOffset_TargetTemperature_HeatPump_HNHT : REAL := 1;
	Controller_HeatPump_HNHT_Permission : FB_CTRL_2POINT;
	Controller_HeatPump_HNHT_Permission_Parameters : ST_CTRL_2POINT_PARAMS;
	fOffset_TargetTemperature_HeatPump_HNHT_Permission : REAL := 1;
	
	//controllers and variables for hnlt and cn linkage
	fOffset_TargetTemperature_HeatPump : REAL;
	Controller_HeatPump : FB_CTRL_2POINT;
	Controller_HeatPump_Parameters : ST_CTRL_2POINT_PARAMS;		

	//clock
	stDefaultParameters_Clock : ST_ClockDefaultParameters := (tTaskCycleTime := GlobalVariables.tCtrlCycleTime_MAIN, tCtrlCycleTime := T#1M);
	Clock : FB_Clock := (ST_DefaultParameters := stDefaultParameters_Clock);
END_VAR

Clock();
AmbientControl();
SetTemperatures();
ControlCN();
ControlHNLT();
ControlHNHT();
ControlHnltCnLinkage();
ControlHnhtHnltLinkage();
SetState();

METHOD AmbientControl : BOOL
VAR_INPUT
END_VAR
//check for heating or cooling mode
IF Clock.stClockState.sintMonth>4 AND Clock.stClockState.sintMonth<10 THEN
	//heating mode
	hnltCnLinkageControl.bHeatingMode := FALSE;
	hnhtCnLinkageControl.bHeatingMode := FALSE;
ELSE
	//cooling mode	
	hnltCnLinkageControl.bHeatingMode := TRUE;
	hnhtCnLinkageControl.bHeatingMode := TRUE;
END_IF
END_METHOD

METHOD ControlCN : BOOL
VAR_INPUT
END_VAR
//set hysteresis parameters for two-point controllers in cooling network
Controller_eChiller_Parameters.fHysteresisRange := 7;
Controller_eChiller_Parameters.tCtrlCycleTime := GlobalVariables.tCtrlCycleTime_MAIN;
Controller_eChiller_Parameters.tTaskCycleTime := GlobalVariables.tTaskCycleTime_MAIN;

//permission to load storage depending on upper hvfa storage temperature
Controller_HVFA_CN_LoadingPermission_Parameters.fHysteresisRange := 1;
Controller_HVFA_CN_LoadingPermission_Parameters.tCtrlCycleTime := GlobalVariables.tCtrlCycleTime_MAIN;
Controller_HVFA_CN_LoadingPermission_Parameters.tTaskCycleTime := GlobalVariables.tTaskCycleTime_MAIN;

//permission to unload storage depending on upper hvfa storage temperature
Controller_HVFA_CN_UnloadingPermission_Parameters.fHysteresisRange := 1;
Controller_HVFA_CN_UnloadingPermission_Parameters.tCtrlCycleTime := GlobalVariables.tCtrlCycleTime_MAIN;
Controller_HVFA_CN_UnloadingPermission_Parameters.tTaskCycleTime := GlobalVariables.tTaskCycleTime_MAIN;

//hysteresis for unloading hvfa storage depending on buffer storage temperature
Controller_Buffer_HVFA_CN_Unloading_Parameters.fHysteresisRange := 2;
Controller_Buffer_HVFA_CN_Unloading_Parameters.tCtrlCycleTime := GlobalVariables.tCtrlCycleTime_MAIN;
Controller_Buffer_HVFA_CN_Unloading_Parameters.tTaskCycleTime := GlobalVariables.tTaskCycleTime_MAIN;

//control eChiller
Controller_eChiller(fSetpointValue := cnState.fMidTemperature,
	fActualValue := fTargetTemperature_CN-fOffset_TargetTemperature_eChiller,
	eMode := eCTRL_MODE_ACTIVE,
	stParams := Controller_eChiller_Parameters);

//control hvfa storage loading permission 
Controller_HVFA_CN_LoadingPermission(fSetpointValue := cnState.fUpperTemperature_ActiveStorage,
	fActualValue := fTargetTemperature_CN-fOffset_TargetTemperature_HVFA_CN_Permission,
	eMode := eCTRL_MODE_ACTIVE,
	stParams := Controller_HVFA_CN_LoadingPermission_Parameters);
	
//control hvfa storage unloading permission 
Controller_HVFA_CN_UnloadingPermission(fSetpointValue := fTargetTemperature_CN-fOffset_TargetTemperature_HVFA_CN_Permission,
	fActualValue := cnState.fLowerTemperature_ActiveStorage,
	eMode := eCTRL_MODE_ACTIVE,
	stParams := Controller_HVFA_CN_UnloadingPermission_Parameters);
	
//unloading permission buffer HVFA
Controller_Buffer_HVFA_CN_Unloading(fSetpointValue := cnState.fMidTemperature,
	fActualValue := fTargetTemperature_CN+fOffset_TargetTemperature_HVFA_CN,
	eMode := eCTRL_MODE_ACTIVE,
	stParams := Controller_Buffer_HVFA_CN_Unloading_Parameters);
	
IF Clock.stClockState.sintMonth>4 AND Clock.stClockState.sintMonth<10 THEN
	cnControl.bSetStatusOn_eChiller := TRUE;
	cnControl.bSetStatusOn_HVFASystem := FALSE;
	cnControl.bLoading_HVFASystem := FALSE;
ELSE
	cnControl.bSetStatusOn_eChiller := Controller_eChiller.bOut;
	cnControl.bSetStatusOn_HVFASystem := (Controller_Buffer_HVFA_CN_Unloading.bOut AND Controller_HVFA_CN_UnloadingPermission.bOut) OR ((cnControl.bSetStatusOn_eChiller) AND NOT Controller_Buffer_HVFA_CN_Unloading.bOut AND Controller_HVFA_CN_LoadingPermission.bOut); 
	cnControl.bLoading_HVFASystem := NOT (Controller_Buffer_HVFA_CN_Unloading.bOut AND Controller_HVFA_CN_UnloadingPermission.bOut);
END_IF

cnControl.bSetStatusOn_eChiller := FALSE; //strategy without eChiller
cnControl.bSetStatusOn_HVFASystem := FALSE;
cnControl.bLoading_HVFASystem := FALSE;


//cnControl.bSetStatusOn_HVFASystem := FALSE;
//cnControl.bLoading_HVFASystem := FALSE;
END_METHOD

METHOD ControlHNHT : BOOL
VAR_INPUT
END_VAR
VAR
END_VAR
//set hysteresis parameters for two-point controllers in high temperature heating network
Controller_CHP_Prioritization_Parameters.fHysteresisRange := 4;
Controller_CHP_Prioritization_Parameters.tCtrlCycleTime := GlobalVariables.tCtrlCycleTime_MAIN;
Controller_CHP_Prioritization_Parameters.tTaskCycleTime := GlobalVariables.tTaskCycleTime_MAIN;

Controller_CHP1_Parameters.tCtrlCycleTime := GlobalVariables.tCtrlCycleTime_MAIN;
Controller_CHP1_Parameters.tTaskCycleTime := GlobalVariables.tTaskCycleTime_MAIN;
Controller_CHP2_Parameters.tCtrlCycleTime := GlobalVariables.tCtrlCycleTime_MAIN;
Controller_CHP2_Parameters.tTaskCycleTime := GlobalVariables.tTaskCycleTime_MAIN;

Controller_CondensingBoiler_Parameters.fHysteresisRange := 12;
Controller_CondensingBoiler_Parameters.tCtrlCycleTime := GlobalVariables.tCtrlCycleTime_MAIN;
Controller_CondensingBoiler_Parameters.tTaskCycleTime := GlobalVariables.tTaskCycleTime_MAIN;

Controller_Buffer_VSI_Unloading_Parameters.fHysteresisRange := 4;
Controller_Buffer_VSI_Unloading_Parameters.tCtrlCycleTime := GlobalVariables.tCtrlCycleTime_MAIN;
Controller_Buffer_VSI_Unloading_Parameters.tTaskCycleTime := GlobalVariables.tTaskCycleTime_MAIN;

Controller_VSI_Unloading_Permission_Parameters.fHysteresisRange := 4;
Controller_VSI_Unloading_Permission_Parameters.tCtrlCycleTime := GlobalVariables.tCtrlCycleTime_MAIN;
Controller_VSI_Unloading_Permission_Parameters.tTaskCycleTime := GlobalVariables.tTaskCycleTime_MAIN;

Controller_VSI_Loading_Permission_Parameters.fHysteresisRange := 4;
Controller_VSI_Loading_Permission_Parameters.tCtrlCycleTime := GlobalVariables.tCtrlCycleTime_MAIN;
Controller_VSI_Loading_Permission_Parameters.tTaskCycleTime := GlobalVariables.tTaskCycleTime_MAIN;

Controller_StaticHeating_Parameters.fHysteresisRange := 4;
Controller_StaticHeating_Parameters.tCtrlCycleTime := GlobalVariables.tCtrlCycleTime_MAIN;
Controller_StaticHeating_Parameters.tTaskCycleTime := GlobalVariables.tTaskCycleTime_MAIN;

Controller_CHP_Prioritization(fSetpointValue := 15,
	fActualValue := ambientState.fOutsideTemperature_Mean,
	eMode := eCTRL_MODE_ACTIVE,
	stParams := Controller_CHP_Prioritization_Parameters);
IF Controller_CHP_Prioritization.bOut THEN
	//prioritize large CHP (CHP2) during cold temperatures
	Controller_CHP1_Parameters.fHysteresisRange := 14;
	Controller_CHP2_Parameters.fHysteresisRange := 12;
	fOffset_TargetTemperature_CHP1 := 1;
	fOffset_TargetTemperature_CHP2 := 0;
ELSE
	//prioritize large CHP (CHP2) during cold temperatures
	Controller_CHP1_Parameters.fHysteresisRange := 12;
	Controller_CHP2_Parameters.fHysteresisRange := 14;	
	fOffset_TargetTemperature_CHP1 := 0;
	fOffset_TargetTemperature_CHP2 := 1;	
END_IF

//start when upper temperature too cold and stop when lower temperature too hot
Controller_CHP1_UpperTemperature(fSetpointValue := fTargetTemperature_HNHT_Heating-fOffset_TargetTemperature_CHP1,
	fActualValue := hnhtState.fUpperTemperature,
	eMode := eCTRL_MODE_ACTIVE,
	stParams := Controller_CHP1_Parameters);
Controller_CHP1_LowerTemperature(fSetpointValue := fTargetTemperature_HNHT_Heating-fOffset_TargetTemperature_CHP1,
	fActualValue := hnhtState.fLowerTemperature,
	eMode := eCTRL_MODE_ACTIVE,
	stParams := Controller_CHP1_Parameters);
Trigger_CHP1_UpperTemperature(CLK := Controller_CHP1_UpperTemperature.bOut);
Trigger_CHP1_LowerTemperature(CLK := Controller_CHP1_LowerTemperature.bOut);
IF Trigger_CHP1_UpperTemperature.Q THEN
	bTrigger_CHP1 := TRUE;
END_IF
IF Trigger_CHP1_LowerTemperature.Q THEN
	bTrigger_CHP1 := FALSE;
END_IF
hnhtControl.bSetStatusOn_CHP1 := Controller_CHP1_UpperTemperature.bOut OR (Controller_CHP1_LowerTemperature.bOut AND bTrigger_CHP1);

//start when upper temperature too cold and stop when lower temperature too hot
Controller_CHP2_UpperTemperature(fSetpointValue := fTargetTemperature_HNHT_Heating-fOffset_TargetTemperature_CHP2,
	fActualValue := hnhtState.fUpperTemperature,
	eMode := eCTRL_MODE_ACTIVE,
	stParams := Controller_CHP2_Parameters);
Controller_CHP2_LowerTemperature(fSetpointValue := fTargetTemperature_HNHT_Heating-fOffset_TargetTemperature_CHP2,
	fActualValue := hnhtState.fLowerTemperature,
	eMode := eCTRL_MODE_ACTIVE,
	stParams := Controller_CHP2_Parameters);
Trigger_CHP2_UpperTemperature(CLK := Controller_CHP2_UpperTemperature.bOut);
Trigger_CHP2_LowerTemperature(CLK := Controller_CHP2_LowerTemperature.bOut);
IF Trigger_CHP2_UpperTemperature.Q THEN
	bTrigger_CHP2 := TRUE;
END_IF
IF Trigger_CHP2_LowerTemperature.Q THEN
	bTrigger_CHP2 := FALSE;
END_IF
hnhtControl.bSetStatusOn_CHP2 := Controller_CHP2_UpperTemperature.bOut OR (Controller_CHP2_LowerTemperature.bOut AND bTrigger_CHP2);

Controller_CondensingBoiler(fSetpointValue := fTargetTemperature_HNHT_Heating,
	fActualValue := hnhtState.fUpperTemperature,
	eMode := eCTRL_MODE_ACTIVE,
	stParams := Controller_CondensingBoiler_Parameters);
hnhtControl.bSetStatusOn_CondensingBoiler := Controller_CondensingBoiler.bOut;

//buffer storage asks VSI for unloading when buffer storage temperature falls below limit
Controller_Buffer_VSI_Unloading(fSetpointValue := fTargetTemperature_HNHT_Heating,
	fActualValue := hnhtState.fUpperTemperature,
	eMode := eCTRL_MODE_ACTIVE,
	stParams := Controller_Buffer_VSI_Unloading_Parameters);

//VSI storage may only be unloaded when upper temperature is between limits for unloading
Controller_VSI_Unloading_Permission(fSetpointValue := hnhtState.fUpperTemperature_ActiveStorage,
	fActualValue := fTargetTemperature_HNHT_Heating,
	eMode := eCTRL_MODE_ACTIVE,
	stParams := Controller_VSI_Unloading_Permission_Parameters);
	
//VSI storage may only be loaded when lower temperature is between limits for loading
Controller_VSI_Loading_Permission(fSetpointValue := fTargetTemperature_HNHT_Heating,
	fActualValue := hnhtState.fLowerTemperature_ActiveStorage,
	eMode := eCTRL_MODE_ACTIVE,
	stParams := Controller_VSI_Loading_Permission_Parameters);
	
hnhtControl.bSetStatusOn_VSIStorage := (Controller_Buffer_VSI_Unloading.bOut AND Controller_VSI_Unloading_Permission.bOut) OR ((hnhtControl.bSetStatusOn_CHP1 OR hnhtControl.bSetStatusOn_CHP2) AND NOT Controller_Buffer_VSI_Unloading.bOut AND Controller_VSI_Loading_Permission.bOut); 
hnhtControl.bLoading_VSISystem := NOT (Controller_Buffer_VSI_Unloading.bOut AND Controller_VSI_Unloading_Permission.bOut);

//condensing boiler is switched if network temperature falls below critical temperature limit
Controller_StaticHeating(fSetpointValue := 15,
	fActualValue := ambientState.fOutsideTemperature,
	eMode := eCTRL_MODE_ACTIVE,
	stParams := Controller_StaticHeating_Parameters);
hnhtControl.bSetStatusOn_StaticHeating := Controller_StaticHeating.bOut;
END_METHOD

METHOD ControlHnhtHnltLinkage : BOOL
VAR_INPUT
END_VAR
Controller_HeatExchanger1_Parameters.fHysteresisRange := 8;
Controller_HeatExchanger1_Parameters.tCtrlCycleTime := GlobalVariables.tCtrlCycleTime_MAIN;
Controller_HeatExchanger1_Parameters.tTaskCycleTime := GlobalVariables.tTaskCycleTime_MAIN;

Controller_HeatPump_HNHT_Parameters.fHysteresisRange := 10;
Controller_HeatPump_HNHT_Parameters.tCtrlCycleTime := GlobalVariables.tCtrlCycleTime_MAIN;
Controller_HeatPump_HNHT_Parameters.tTaskCycleTime := GlobalVariables.tTaskCycleTime_MAIN;

Controller_HeatPump_HNHT_Permission_Parameters.fHysteresisRange := 4;
Controller_HeatPump_HNHT_Permission_Parameters.tCtrlCycleTime := GlobalVariables.tCtrlCycleTime_MAIN;
Controller_HeatPump_HNHT_Permission_Parameters.tTaskCycleTime := GlobalVariables.tTaskCycleTime_MAIN;

//control heat exchanger 1
Controller_HeatExchanger1(fSetpointValue := fTargetTemperature_HNLT_Heating-fOffset_TargetTemperature_HeatExchanger1,
	fActualValue := hnltState.fMidTemperature,
	eMode := eCTRL_MODE_ACTIVE,
	stParams := Controller_HeatExchanger1_Parameters);
hnhtHnltLinkageControl.bSetStatusOn_HeatExchanger1 := Controller_HeatExchanger1.bOut;

//control heat pump hnht
Controller_HeatPump_HNHT(fSetpointValue := fTargetTemperature_HNHT_Heating+fOffset_TargetTemperature_HeatPump_HNHT,
	fActualValue := hnhtState.fUpperTemperature,
	eMode := eCTRL_MODE_ACTIVE,
	stParams := Controller_HeatPump_HNHT_Parameters);
	
Controller_HeatPump_HNHT_Permission(fSetpointValue := hnltState.fMidTemperature,
	fActualValue := fTargetTemperature_HNLT_Cooling+fOffset_TargetTemperature_HeatPump_HNHT_Permission,
	eMode := eCTRL_MODE_ACTIVE,
	stParams := Controller_HeatPump_HNHT_Permission_Parameters);	
	
// HP currently only able to reach 65°C flow temperature (hard-coded HP-internal)
// IF localSetParameters.bProductionModeActivated THEN
// 	hnhtHnltLinkageControl.bSetStatusOn_HeatPump := FALSE;
// ELSE
// 	hnhtHnltLinkageControl.bSetStatusOn_HeatPump := Controller_HeatPump_HNHT.bOut AND Controller_HeatPump_HNHT_Permission.bOut;
// END_IF

// When using a heating target temp of 60 °C in production mode the heat pump can be used in both operating modes
hnhtHnltLinkageControl.bSetStatusOn_HeatPump := Controller_HeatPump_HNHT.bOut AND Controller_HeatPump_HNHT_Permission.bOut;
END_METHOD

METHOD ControlHNLT : BOOL
VAR_INPUT
END_VAR
//set hysteresis parameters for two-point controllers in cooling network
Controller_OuterCapillaryTubeMats_Parameters.fHysteresisRange := 6;
Controller_OuterCapillaryTubeMats_Parameters.tCtrlCycleTime := GlobalVariables.tCtrlCycleTime_MAIN;
Controller_OuterCapillaryTubeMats_Parameters.tTaskCycleTime := GlobalVariables.tTaskCycleTime_MAIN;

Controller_OuterCapillaryTubeMats_Permission_Parameters.fHysteresisRange := 6;
Controller_OuterCapillaryTubeMats_Permission_Parameters.tCtrlCycleTime := GlobalVariables.tCtrlCycleTime_MAIN;
Controller_OuterCapillaryTubeMats_Permission_Parameters.tTaskCycleTime := GlobalVariables.tTaskCycleTime_MAIN;


//control strategy for cooling network - fSetpointValue and fActualValue are changed for cooling applications
Controller_OuterCapillaryTubeMats(fSetpointValue := hnltState.fMidTemperature,
	fActualValue := fTargetTemperature_HNLT_Cooling+fOffset_TargetTemperature_OuterCapillaryTubeMats_Cooling,
	eMode := eCTRL_MODE_ACTIVE,
	stParams := Controller_OuterCapillaryTubeMats_Parameters);

//permission controller to ensure that network ist not heated up if ambient temperature is too high
Controller_OuterCapillaryTubeMats_Permission(fSetpointValue := fTargetTemperature_HNLT_Cooling-fOffset_OuterCapillaryTubeMats_Permission,
	fActualValue := ambientState.fOutsideTemperature,
	eMode := eCTRL_MODE_ACTIVE,
	stParams := Controller_OuterCapillaryTubeMats_Permission_Parameters);

//control hvfa storage
//set hysteresis parameters for two-point controllers in low temperature heating network

Controller_Buffer_HVFA_HNLT_HVFAUnloading_Parameters.fHysteresisRange := 6;
Controller_Buffer_HVFA_HNLT_HVFAUnloading_Parameters.tCtrlCycleTime := GlobalVariables.tCtrlCycleTime_MAIN;
Controller_Buffer_HVFA_HNLT_HVFAUnloading_Parameters.tTaskCycleTime := GlobalVariables.tTaskCycleTime_MAIN;

Controller_Buffer_HVFA_HNLT_HVFALoading_Parameters.fHysteresisRange := 4;
Controller_Buffer_HVFA_HNLT_HVFALoading_Parameters.tCtrlCycleTime := GlobalVariables.tCtrlCycleTime_MAIN;
Controller_Buffer_HVFA_HNLT_HVFALoading_Parameters.tTaskCycleTime := GlobalVariables.tTaskCycleTime_MAIN;

Controller_HVFA_HNLT_Recooling_Parameters.fHysteresisRange := 4;
Controller_HVFA_HNLT_Recooling_Parameters.tCtrlCycleTime := GlobalVariables.tCtrlCycleTime_MAIN;
Controller_HVFA_HNLT_Recooling_Parameters.tTaskCycleTime := GlobalVariables.tTaskCycleTime_MAIN;

Controller_HVFA_HNLT_HVFAUnloadingPermission_Parameters.fHysteresisRange := 4;
Controller_HVFA_HNLT_HVFAUnloadingPermission_Parameters.tCtrlCycleTime := GlobalVariables.tCtrlCycleTime_MAIN;
Controller_HVFA_HNLT_HVFAUnloadingPermission_Parameters.tTaskCycleTime := GlobalVariables.tTaskCycleTime_MAIN;

Controller_HVFA_HNLT_HVFALoadingPermission_Parameters.fHysteresisRange := 4;
Controller_HVFA_HNLT_HVFALoadingPermission_Parameters.tCtrlCycleTime := GlobalVariables.tCtrlCycleTime_MAIN;
Controller_HVFA_HNLT_HVFALoadingPermission_Parameters.tTaskCycleTime := GlobalVariables.tTaskCycleTime_MAIN;

//buffer storage asks HVFA_HNLT for unloading when buffer storage temperature falls below limit
Controller_Buffer_HVFA_HNLT_HVFAUnloading(fSetpointValue := fTargetTemperature_HNLT_Heating-fOffset_TargetTemperature_HVFA_HNLT_Heating,
	fActualValue := hnltState.fMidTemperature,
	eMode := eCTRL_MODE_ACTIVE,
	stParams := Controller_Buffer_HVFA_HNLT_HVFAUnloading_Parameters);
	
//buffer storage asks HVFA_HNLT for loading when buffer storage temperature rises above limit
Controller_Buffer_HVFA_HNLT_HVFALoading(fSetpointValue := hnltState.fMidTemperature,
	fActualValue := fTargetTemperature_HNLT_Cooling,
	eMode := eCTRL_MODE_ACTIVE,
	stParams := Controller_Buffer_HVFA_HNLT_HVFALoading_Parameters);

//hvfa storage may only be unloaded when upper temperature is between limits for unloading
Controller_HVFA_HNLT_HVFAUnloadingPermission(fSetpointValue := hnltState.fLowerTemperature_ActiveStorage,
	fActualValue := fTargetTemperature_HNLT_Heating,
	eMode := eCTRL_MODE_ACTIVE,
	stParams := Controller_HVFA_HNLT_HVFAUnloadingPermission_Parameters);
	
//hvfa storage may only be loaded when lower temperature is between limits for loading
Controller_HVFA_HNLT_HVFALoadingPermission(fSetpointValue := fTargetTemperature_HNLT_Cooling,
	fActualValue := hnltState.fLowerTemperature_ActiveStorage,
	eMode := eCTRL_MODE_ACTIVE,
	stParams := Controller_HVFA_HNLT_HVFALoadingPermission_Parameters);

//enable hvfa recooling during low temperature times in summer months	
Controller_HVFA_HNLT_Recooling(fSetpointValue := hnltState.fLowerTemperature_ActiveStorage,
	fActualValue := fTargetTemperature_HNLT_Cooling-fOffset_HVFA_HNLT_Recooling,
	eMode := eCTRL_MODE_ACTIVE,
	stParams := Controller_HVFA_HNLT_Recooling_Parameters);
	
IF hnltCnLinkageControl.bHeatingMode THEN
	hnltControl.bSetStatusOn_HVFASystem := (Controller_HVFA_HNLT_HVFALoadingPermission.bOut AND Controller_Buffer_HVFA_HNLT_HVFALoading.bOut) OR (Controller_HVFA_HNLT_HVFAUnloadingPermission.bOut AND Controller_Buffer_HVFA_HNLT_HVFAUnloading.bOut);
	hnltControl.bLoading_HVFASystem := Controller_HVFA_HNLT_HVFALoadingPermission.bOut AND Controller_Buffer_HVFA_HNLT_HVFALoading.bOut;
	hnltControl.bSetStatusOn_OuterCapillaryTubeMats := Controller_OuterCapillaryTubeMats.bOut AND Controller_OuterCapillaryTubeMats_Permission.bOut;
ELSE
	hnltControl.bSetStatusOn_HVFASystem := ((Controller_HVFA_HNLT_HVFALoadingPermission.bOut AND Controller_Buffer_HVFA_HNLT_HVFALoading.bOut) OR (Controller_HVFA_HNLT_HVFAUnloadingPermission.bOut AND Controller_Buffer_HVFA_HNLT_HVFAUnloading.bOut)) OR (Controller_HVFA_HNLT_Recooling.bOut AND Controller_OuterCapillaryTubeMats_Permission.bOut);
	hnltControl.bLoading_HVFASystem := Controller_HVFA_HNLT_HVFALoadingPermission.bOut AND Controller_Buffer_HVFA_HNLT_HVFALoading.bOut;
	hnltControl.bSetStatusOn_OuterCapillaryTubeMats := (Controller_OuterCapillaryTubeMats.bOut AND Controller_OuterCapillaryTubeMats_Permission.bOut) OR (Controller_HVFA_HNLT_Recooling.bOut AND Controller_OuterCapillaryTubeMats_Permission.bOut);
END_IF
END_METHOD

METHOD ControlHnltCnLinkage : BOOL
VAR_INPUT
END_VAR
//set hysteresis parameters for hnlt cn linkage systems
fOffset_TargetTemperature_HeatPump := 0;
Controller_HeatPump_Parameters.fHysteresisRange := 4;
Controller_HeatPump_Parameters.tCtrlCycleTime := GlobalVariables.tCtrlCycleTime_MAIN;
Controller_HeatPump_Parameters.tTaskCycleTime := GlobalVariables.tTaskCycleTime_MAIN;
	
//control heat pump depending on heating demand in hnlt

Controller_HeatPump(fSetpointValue := cnState.fMidTemperature,
	fActualValue := fTargetTemperature_CN,
	eMode := eCTRL_MODE_ACTIVE,
	stParams := Controller_HeatPump_Parameters);
	
hnltCnLinkageControl.bSetStatusOn_HeatPump := Controller_HeatPump.bOut;

hnltCnLinkageControl.fTargetTemperature_ProductionHall := localDefaultParameters.fTargetTemperature_ProductionHall;

hnltCnLinkageControl.bSetStatusOn_InnerCapillaryTubeMats := FALSE; //turn off cooling when eChiller is not available
hnltCnLinkageControl.bSetStatusOn_UnderfloorHeating := FALSE; //turn off cooling when eChiller is not available
END_METHOD

METHOD SetState : BOOL
VAR_INPUT
END_VAR
localState.fTargetTemperature_HNHT_Heating := fTargetTemperature_HNHT_Heating;
localState.fTargetTemperature_HNHT_Cooling := fTargetTemperature_HNHT_Cooling;
localState.fTargetTemperature_HNLT_Heating := fTargetTemperature_HNLT_Heating;
localState.fTargetTemperature_HNLT_Cooling := fTargetTemperature_HNLT_Cooling;
localState.fTargetTemperature_CN := fTargetTemperature_CN;
localState.fTargetTemperature_ProductionHall := localDefaultParameters.fTargetTemperature_ProductionHall;

localState.aTemperatureLimits_HNHT := aTemperatureLimits_HNHT;
localState.aTemperatureLimits_HNLT := aTemperatureLimits_HNLT;
localState.aTemperatureLimits_CN := aTemperatureLimits_CN;	

localState.fFeedTemperature_HNHT := fTargetTemperature_HNHT_Heating+localDefaultParameters.fOffset_FeedTemperature_HNHT;
localState.fFeedTemperature_HNLT_Heating := fTargetTemperature_HNLT_Heating+localDefaultParameters.fOffset_FeedTemperature_HNLT_Heating;
localState.fFeedTemperature_HNLT_Cooling := fTargetTemperature_HNLT_Cooling-localDefaultParameters.fOffset_FeedTemperature_HNLT_Cooling;
localState.fFeedTemperature_CN := fTargetTemperature_CN-localDefaultParameters.fOffset_FeedTemperature_CN;
END_METHOD

METHOD SetTemperatures : BOOL
VAR_INPUT
END_VAR
//set internal variables depending on prodution mode
IF localSetParameters.bProductionModeActivated THEN
	IF Clock.stClockState.sintMonth>4 AND Clock.stClockState.sintMonth<10 THEN	
		fTargetTemperature_CN := localDefaultParameters.fTargetTemperature_CN_ProductionMode_Summer;
	ELSE
		fTargetTemperature_CN := localDefaultParameters.fTargetTemperature_CN_ProductionMode_Winter;
	END_IF
	fTargetTemperature_HNLT_Heating := localDefaultParameters.fTargetTemperature_HNLT_Heating_ProductionMode;
	fTargetTemperature_HNLT_Cooling := localDefaultParameters.fTargetTemperature_HNLT_Cooling_ProductionMode;
	fTargetTemperature_HNHT_Heating := localDefaultParameters.fTargetTemperature_HNHT_Heating_ProductionMode;
	fTargetTemperature_HNHT_Cooling := localDefaultParameters.fTargetTemperature_HNHT_Cooling_ProductionMode;
	aTemperatureLimits_CN := localDefaultParameters.aTemperatureLimits_CN_ProductionMode;
	aTemperatureLimits_HNLT := localDefaultParameters.aTemperatureLimits_HNLT_ProductionMode;
	aTemperatureLimits_HNHT := localDefaultParameters.aTemperatureLimits_HNHT_ProductionMode;

ELSE
	IF Clock.stClockState.sintMonth>4 AND Clock.stClockState.sintMonth<10 THEN	
		fTargetTemperature_CN := localDefaultParameters.fTargetTemperature_CN_Summer;
	ELSE
		fTargetTemperature_CN := localDefaultParameters.fTargetTemperature_CN_Winter;
	END_IF
	fTargetTemperature_HNLT_Heating := localDefaultParameters.fTargetTemperature_HNLT_Heating;
	fTargetTemperature_HNLT_Cooling := localDefaultParameters.fTargetTemperature_HNLT_Cooling;
	fTargetTemperature_HNHT_Heating := localDefaultParameters.fTargetTemperature_HNHT_Heating;
	fTargetTemperature_HNHT_Cooling := localDefaultParameters.fTargetTemperature_HNHT_Cooling;
	aTemperatureLimits_CN := localDefaultParameters.aTemperatureLimits_CN;
	aTemperatureLimits_HNLT := localDefaultParameters.aTemperatureLimits_HNLT;
	aTemperatureLimits_HNHT := localDefaultParameters.aTemperatureLimits_HNHT;
END_IF

//set feed temperatures
hnhtControl.fFeedTemperature := fTargetTemperature_HNHT_Heating+localDefaultParameters.fOffset_FeedTemperature_HNHT;
hnltControl.fFeedTemperature_Heating := fTargetTemperature_HNLT_Heating+localDefaultParameters.fOffset_FeedTemperature_HNLT_Heating;
hnltControl.fFeedTemperature_Cooling := fTargetTemperature_HNLT_Cooling-localDefaultParameters.fOffset_FeedTemperature_HNLT_Cooling;
cnControl.fFeedTemperature := fTargetTemperature_CN-localDefaultParameters.fOffset_FeedTemperature_CN;
hnhtHnltLinkageControl.fFeedTemperature_HNHT := hnhtControl.fFeedTemperature;
hnhtHnltLinkageControl.fFeedTemperature_HNLT_Heating := hnltControl.fFeedTemperature_Heating;
hnhtHnltLinkageControl.fFeedTemperature_HNLT_Cooling := hnltControl.fFeedTemperature_Cooling;
hnltCnLinkageControl.fFeedTemperature_CN := cnControl.fFeedTemperature;
hnltCnLinkageControl.fFeedTemperature_HNLT_Heating := hnltControl.fFeedTemperature_Heating;
hnltCnLinkageControl.fFeedTemperature_HNLT_Cooling := hnltControl.fFeedTemperature_Cooling;

//set algorithm permission depending on production mode to control structs
CN_Check(fInput := cnState.fMidTemperature,
	fLowerLimit := aTemperatureLimits_CN[1],
	fUpperLimit := aTemperatureLimits_CN[2]);
cnControl.bAlgorithmPermission := CN_Check.bPermission;
	
HNLT_Check(fInput := hnltState.fMidTemperature,
	fLowerLimit := aTemperatureLimits_HNLT[1],
	fUpperLimit := aTemperatureLimits_HNLT[2]);
hnltControl.bAlgorithmPermission := HNLT_Check.bPermission;
	
HNHT_Check(fInput := hnhtState.fMidTemperature,
	fLowerLimit := aTemperatureLimits_HNHT[1],
	fUpperLimit := aTemperatureLimits_HNHT[2]);	
hnhtControl.bAlgorithmPermission := HNHT_Check.bPermission;
	
hnltCnLinkageControl.bAlgorithmPermission_CN := cnControl.bAlgorithmPermission;
hnltCnLinkageControl.bAlgorithmPermission_HNLT := hnltControl.bAlgorithmPermission;
hnhtHnltLinkageControl.bAlgorithmPermission_HNHT := hnhtControl.bAlgorithmPermission;
hnhtHnltLinkageControl.bAlgorithmPermission_HNLT := hnltControl.bAlgorithmPermission;
hnhtCnLinkageControl.bAlgorithmPermission_CN := cnControl.bAlgorithmPermission;
hnhtCnLinkageControl.bAlgorithmPermission_HNHT := hnhtControl.bAlgorithmPermission;
END_METHOD

END_FUNCTION_BLOCK

// ---- POUs/06 Strategy/FB_StrategyController_NoStorages.TcPOU
FUNCTION_BLOCK FB_StrategyController_NoStorages
VAR_INPUT
	ambientState : ST_AmbientState;
	
	//actual temperatures in thermal networks
	cnState : ST_ThermalNetworkState;
	hnltState : ST_ThermalNetworkState;
	hnhtState : ST_ThermalNetworkState;
END_VAR
VAR_OUTPUT	
	cnControl : ST_CoolingNetworkControl;
	hnltControl : ST_HeatingNetworkLowTemperatureControl;	
	hnhtControl : ST_HeatingNetworkHighTemperatureControl;
	hnltCnLinkageControl : ST_HnltCnLinkageControl;
	hnhtHnltLinkageControl : ST_HnhtHnltLinkageControl;
	hnhtCnLinkageControl : ST_HnhtCnLinkageControl;
END_VAR
VAR
	{attribute 'OPC.UA.DA' := '1'}
	localSetParameters : ST_StrategySetParameters;	
	{attribute 'OPC.UA.DA' := '1'}
	localState : ST_StrategyState;	

	//default parameters
	localDefaultParameters : ST_StrategyDefaultParameters;

	//internal variables
	fTargetTemperature_HNHT_Heating : REAL;
	fTargetTemperature_HNHT_Cooling : REAL;
	fTargetTemperature_HNLT_Cooling : REAL;
	fTargetTemperature_HNLT_Heating : REAL;
	fTargetTemperature_CN : REAL;
	aTemperatureLimits_HNHT : ARRAY[1..2] OF REAL;
	aTemperatureLimits_HNLT : ARRAY[1..2] OF REAL;
	aTemperatureLimits_CN : ARRAY[1..2] OF REAL;
	stHNHTCheckDefaultParameters : ST_RangeCheckDefaultParameters := (tTaskCycleTime := GlobalVariables.tCtrlCycleTime_MAIN, tCtrlCycleTime := GlobalVariables.tCtrlCycleTime_MAIN, fRestoreDifference := 5);
	HNHT_Check : FB_RangeCheck := (ST_DefaultParameters := stHNHTCheckDefaultParameters);
	stHNLTCheckDefaultParameters : ST_RangeCheckDefaultParameters := (tTaskCycleTime := GlobalVariables.tCtrlCycleTime_MAIN, tCtrlCycleTime := GlobalVariables.tCtrlCycleTime_MAIN, fRestoreDifference := 5);
	HNLT_Check : FB_RangeCheck := (ST_DefaultParameters := stHNLTCheckDefaultParameters);
	stCNCheckDefaultParameters : ST_RangeCheckDefaultParameters := (tTaskCycleTime := GlobalVariables.tCtrlCycleTime_MAIN, tCtrlCycleTime := GlobalVariables.tCtrlCycleTime_MAIN, fRestoreDifference := 2);
	CN_Check : FB_RangeCheck := (ST_DefaultParameters := stCNCheckDefaultParameters);
	
	
	//controller and variables for high temperature heating network
	fOffset_TargetTemperature_CHP1 : REAL; //not fixed, switches depending on ambient temperature -> see method: ControlHNHT
	fOffset_TargetTemperature_CHP2 : REAL; //not fixed, switches depending on ambient temperature -> see method: ControlHNHT
	Controller_CHP_Prioritization : FB_CTRL_2POINT;
	Controller_CHP_Prioritization_Parameters : ST_CTRL_2POINT_PARAMS;	
	Controller_CHP1_UpperTemperature : FB_CTRL_2POINT; //check upper temperature for turning on chp
	Controller_CHP1_LowerTemperature : FB_CTRL_2POINT; //check lower temperature for turning off chp
	Controller_CHP1_Parameters : ST_CTRL_2POINT_PARAMS;	
	Trigger_CHP1_UpperTemperature : F_TRIG;
	Trigger_CHP1_LowerTemperature : F_TRIG;
	bTrigger_CHP1 : BOOL;
	Controller_CHP2_UpperTemperature : FB_CTRL_2POINT;
	Controller_CHP2_LowerTemperature : FB_CTRL_2POINT;
	Controller_CHP2_Parameters : ST_CTRL_2POINT_PARAMS;
	Trigger_CHP2_UpperTemperature : F_TRIG;
	Trigger_CHP2_LowerTemperature : F_TRIG;
	bTrigger_CHP2 : BOOL;
	Controller_CondensingBoiler : FB_CTRL_2POINT;
	Controller_CondensingBoiler_Parameters : ST_CTRL_2POINT_PARAMS;
	Controller_StaticHeating : FB_CTRL_2POINT;
	Controller_StaticHeating_Parameters : ST_CTRL_2POINT_PARAMS;
	
	//controllers and variables for low temperature heating network
	Controller_OuterCapillaryTubeMats : FB_CTRL_2POINT;
	Controller_OuterCapillaryTubeMats_Parameters : ST_CTRL_2POINT_PARAMS;
	Controller_OuterCapillaryTubeMats_Permission : FB_CTRL_2POINT;
	Controller_OuterCapillaryTubeMats_Permission_Parameters : ST_CTRL_2POINT_PARAMS;
	fOffset_TargetTemperature_OuterCapillaryTubeMats_Cooling : REAL := 1;	
	fOffset_OuterCapillaryTubeMats_Permission : REAL := 10;	
	
	//controllers and variables for cooling network
	fOffset_TargetTemperature_eChiller : REAL := 0.5;	
	fOffset_TargetTemperature_HVFA_CN : REAL := 1;
	fOffset_TargetTemperature_HVFA_CN_Permission : REAL := 2.5;
	Controller_eChiller : FB_CTRL_2POINT;
	Controller_eChiller_Parameters : ST_CTRL_2POINT_PARAMS;	

	//controllers and variables for hnht and hnlt linkage
	Controller_HeatExchanger1 : FB_CTRL_2POINT;
	Controller_HeatExchanger1_Parameters : ST_CTRL_2POINT_PARAMS;
	fOffset_TargetTemperature_HeatExchanger1 : REAL := 2;
	Controller_HeatPump_HNHT : FB_CTRL_2POINT;
	Controller_HeatPump_HNHT_Parameters : ST_CTRL_2POINT_PARAMS;
	fOffset_TargetTemperature_HeatPump_HNHT : REAL := 1;
	Controller_HeatPump_HNHT_Permission : FB_CTRL_2POINT;
	Controller_HeatPump_HNHT_Permission_Parameters : ST_CTRL_2POINT_PARAMS;
	fOffset_TargetTemperature_HeatPump_HNHT_Permission : REAL := 1;
	
	//controllers and variables for hnlt and cn linkage
	fOffset_TargetTemperature_HeatPump : REAL;
	fOffset_TargetTemperature_HeatPump_Permission : REAL;
	Controller_HeatPump : FB_CTRL_2POINT;
	Controller_HeatPump_Parameters : ST_CTRL_2POINT_PARAMS;	
	Controller_HeatPump_Permission : FB_CTRL_2POINT;
	Controller_HeatPump_Permission_Parameters : ST_CTRL_2POINT_PARAMS;	

	//clock
	stDefaultParameters_Clock : ST_ClockDefaultParameters := (tTaskCycleTime := GlobalVariables.tCtrlCycleTime_MAIN, tCtrlCycleTime := T#1M);
	Clock : FB_Clock := (ST_DefaultParameters := stDefaultParameters_Clock);
END_VAR

Clock();
AmbientControl();
SetTemperatures();
ControlCN();
ControlHNLT();
ControlHNHT();
ControlHnltCnLinkage();
ControlHnhtHnltLinkage();
SetState();

METHOD AmbientControl : BOOL
VAR_INPUT
END_VAR
//check for heating or cooling mode
IF Clock.stClockState.sintMonth>4 AND Clock.stClockState.sintMonth<10 THEN
	//heating mode
	hnltCnLinkageControl.bHeatingMode := FALSE;
	hnhtCnLinkageControl.bHeatingMode := FALSE;
ELSE
	//cooling mode	
	hnltCnLinkageControl.bHeatingMode := TRUE;
	hnhtCnLinkageControl.bHeatingMode := TRUE;
END_IF
END_METHOD

METHOD ControlCN : BOOL
VAR_INPUT
END_VAR
//set hysteresis parameters for two-point controllers in cooling network
Controller_eChiller_Parameters.fHysteresisRange := 7;
Controller_eChiller_Parameters.tCtrlCycleTime := GlobalVariables.tCtrlCycleTime_MAIN;
Controller_eChiller_Parameters.tTaskCycleTime := GlobalVariables.tTaskCycleTime_MAIN;


//control eChiller
Controller_eChiller(fSetpointValue := cnState.fMidTemperature,
	fActualValue := fTargetTemperature_CN-fOffset_TargetTemperature_eChiller,
	eMode := eCTRL_MODE_ACTIVE,
	stParams := Controller_eChiller_Parameters);

cnControl.bSetStatusOn_eChiller := Controller_eChiller.bOut;	

cnControl.bSetStatusOn_HVFASystem := FALSE;
cnControl.bLoading_HVFASystem := FALSE;
END_METHOD

METHOD ControlHNHT : BOOL
VAR_INPUT
END_VAR
VAR
END_VAR
//set hysteresis parameters for two-point controllers in high temperature heating network
Controller_CHP_Prioritization_Parameters.fHysteresisRange := 4;
Controller_CHP_Prioritization_Parameters.tCtrlCycleTime := GlobalVariables.tCtrlCycleTime_MAIN;
Controller_CHP_Prioritization_Parameters.tTaskCycleTime := GlobalVariables.tTaskCycleTime_MAIN;

Controller_CHP1_Parameters.tCtrlCycleTime := GlobalVariables.tCtrlCycleTime_MAIN;
Controller_CHP1_Parameters.tTaskCycleTime := GlobalVariables.tTaskCycleTime_MAIN;
Controller_CHP2_Parameters.tCtrlCycleTime := GlobalVariables.tCtrlCycleTime_MAIN;
Controller_CHP2_Parameters.tTaskCycleTime := GlobalVariables.tTaskCycleTime_MAIN;

Controller_CondensingBoiler_Parameters.fHysteresisRange := 12;
Controller_CondensingBoiler_Parameters.tCtrlCycleTime := GlobalVariables.tCtrlCycleTime_MAIN;
Controller_CondensingBoiler_Parameters.tTaskCycleTime := GlobalVariables.tTaskCycleTime_MAIN;

Controller_StaticHeating_Parameters.fHysteresisRange := 4;
Controller_StaticHeating_Parameters.tCtrlCycleTime := GlobalVariables.tCtrlCycleTime_MAIN;
Controller_StaticHeating_Parameters.tTaskCycleTime := GlobalVariables.tTaskCycleTime_MAIN;

//operating hours of chp1 should be included
Controller_CHP_Prioritization(fSetpointValue := 15,
	fActualValue := ambientState.fOutsideTemperature_Mean,
	eMode := eCTRL_MODE_ACTIVE,
	stParams := Controller_CHP_Prioritization_Parameters);
IF Controller_CHP_Prioritization.bOut THEN
	//prioritize large CHP (CHP2) during cold temperatures
	Controller_CHP1_Parameters.fHysteresisRange := 14;
	Controller_CHP2_Parameters.fHysteresisRange := 12;
	fOffset_TargetTemperature_CHP1 := 1;
	fOffset_TargetTemperature_CHP2 := 0;
ELSE
	//prioritize large CHP (CHP2) during cold temperatures
	Controller_CHP1_Parameters.fHysteresisRange := 12;
	Controller_CHP2_Parameters.fHysteresisRange := 14;	
	fOffset_TargetTemperature_CHP1 := 0;
	fOffset_TargetTemperature_CHP2 := 1;	
END_IF

//start when upper temperature too cold and stop when lower temperature too hot
Controller_CHP1_UpperTemperature(fSetpointValue := fTargetTemperature_HNHT_Heating-fOffset_TargetTemperature_CHP1,
	fActualValue := hnhtState.fUpperTemperature,
	eMode := eCTRL_MODE_ACTIVE,
	stParams := Controller_CHP1_Parameters);
Controller_CHP1_LowerTemperature(fSetpointValue := fTargetTemperature_HNHT_Heating-fOffset_TargetTemperature_CHP1,
	fActualValue := hnhtState.fLowerTemperature,
	eMode := eCTRL_MODE_ACTIVE,
	stParams := Controller_CHP1_Parameters);
Trigger_CHP1_UpperTemperature(CLK := Controller_CHP1_UpperTemperature.bOut);
Trigger_CHP1_LowerTemperature(CLK := Controller_CHP1_LowerTemperature.bOut);
IF Trigger_CHP1_UpperTemperature.Q THEN
	bTrigger_CHP1 := TRUE;
END_IF
IF Trigger_CHP1_LowerTemperature.Q THEN
	bTrigger_CHP1 := FALSE;
END_IF
hnhtControl.bSetStatusOn_CHP1 := Controller_CHP1_UpperTemperature.bOut OR (Controller_CHP1_LowerTemperature.bOut AND bTrigger_CHP1);

//start when upper temperature too cold and stop when lower temperature too hot
Controller_CHP2_UpperTemperature(fSetpointValue := fTargetTemperature_HNHT_Heating-fOffset_TargetTemperature_CHP2,
	fActualValue := hnhtState.fUpperTemperature,
	eMode := eCTRL_MODE_ACTIVE,
	stParams := Controller_CHP2_Parameters);
Controller_CHP2_LowerTemperature(fSetpointValue := fTargetTemperature_HNHT_Heating-fOffset_TargetTemperature_CHP2,
	fActualValue := hnhtState.fLowerTemperature,
	eMode := eCTRL_MODE_ACTIVE,
	stParams := Controller_CHP2_Parameters);
Trigger_CHP2_UpperTemperature(CLK := Controller_CHP2_UpperTemperature.bOut);
Trigger_CHP2_LowerTemperature(CLK := Controller_CHP2_LowerTemperature.bOut);
IF Trigger_CHP2_UpperTemperature.Q THEN
	bTrigger_CHP2 := TRUE;
END_IF
IF Trigger_CHP2_LowerTemperature.Q THEN
	bTrigger_CHP2 := FALSE;
END_IF
hnhtControl.bSetStatusOn_CHP2 := Controller_CHP2_UpperTemperature.bOut OR (Controller_CHP2_LowerTemperature.bOut AND bTrigger_CHP2);

Controller_CondensingBoiler(fSetpointValue := fTargetTemperature_HNHT_Heating,
	fActualValue := hnhtState.fUpperTemperature,
	eMode := eCTRL_MODE_ACTIVE,
	stParams := Controller_CondensingBoiler_Parameters);
hnhtControl.bSetStatusOn_CondensingBoiler := Controller_CondensingBoiler.bOut;

// turn VSI off
hnhtControl.bSetStatusOn_VSIStorage := FALSE;
hnhtControl.bLoading_VSISystem := FALSE;

//condensing boiler is switched if network temperature falls below critical temperature limit
Controller_StaticHeating(fSetpointValue := 15,
	fActualValue := ambientState.fOutsideTemperature,
	eMode := eCTRL_MODE_ACTIVE,
	stParams := Controller_StaticHeating_Parameters);
hnhtControl.bSetStatusOn_StaticHeating := Controller_StaticHeating.bOut;
END_METHOD

METHOD ControlHnhtHnltLinkage : BOOL
VAR_INPUT
END_VAR
Controller_HeatExchanger1_Parameters.fHysteresisRange := 8;
Controller_HeatExchanger1_Parameters.tCtrlCycleTime := GlobalVariables.tCtrlCycleTime_MAIN;
Controller_HeatExchanger1_Parameters.tTaskCycleTime := GlobalVariables.tTaskCycleTime_MAIN;

Controller_HeatPump_HNHT_Parameters.fHysteresisRange := 10;
Controller_HeatPump_HNHT_Parameters.tCtrlCycleTime := GlobalVariables.tCtrlCycleTime_MAIN;
Controller_HeatPump_HNHT_Parameters.tTaskCycleTime := GlobalVariables.tTaskCycleTime_MAIN;

Controller_HeatPump_HNHT_Permission_Parameters.fHysteresisRange := 4;
Controller_HeatPump_HNHT_Permission_Parameters.tCtrlCycleTime := GlobalVariables.tCtrlCycleTime_MAIN;
Controller_HeatPump_HNHT_Permission_Parameters.tTaskCycleTime := GlobalVariables.tTaskCycleTime_MAIN;

//control heat exchanger 1
Controller_HeatExchanger1(fSetpointValue := fTargetTemperature_HNLT_Heating-fOffset_TargetTemperature_HeatExchanger1,
	fActualValue := hnltState.fMidTemperature,
	eMode := eCTRL_MODE_ACTIVE,
	stParams := Controller_HeatExchanger1_Parameters);
hnhtHnltLinkageControl.bSetStatusOn_HeatExchanger1 := Controller_HeatExchanger1.bOut;

//control heat pump hnht
Controller_HeatPump_HNHT(fSetpointValue := fTargetTemperature_HNHT_Heating+fOffset_TargetTemperature_HeatPump_HNHT,
	fActualValue := hnhtState.fUpperTemperature,
	eMode := eCTRL_MODE_ACTIVE,
	stParams := Controller_HeatPump_HNHT_Parameters);
	
Controller_HeatPump_HNHT_Permission(fSetpointValue := hnltState.fMidTemperature,
	fActualValue := fTargetTemperature_HNLT_Cooling+fOffset_TargetTemperature_HeatPump_HNHT_Permission,
	eMode := eCTRL_MODE_ACTIVE,
	stParams := Controller_HeatPump_HNHT_Permission_Parameters);	
	
// HP currently only able to reach 65°C flow temperature (hard-coded HP-internal)
// IF localSetParameters.bProductionModeActivated THEN
// 	hnhtHnltLinkageControl.bSetStatusOn_HeatPump := FALSE;
// ELSE
// 	hnhtHnltLinkageControl.bSetStatusOn_HeatPump := Controller_HeatPump_HNHT.bOut AND Controller_HeatPump_HNHT_Permission.bOut;
//END_IF

// When using a heating target temp of 60 °C in production mode the heat pump can be used in both operating modes
hnhtHnltLinkageControl.bSetStatusOn_HeatPump := Controller_HeatPump_HNHT.bOut AND Controller_HeatPump_HNHT_Permission.bOut;
END_METHOD

METHOD ControlHNLT : BOOL
VAR_INPUT
END_VAR
//set hysteresis parameters for two-point controllers in cooling network
Controller_OuterCapillaryTubeMats_Parameters.fHysteresisRange := 6;
Controller_OuterCapillaryTubeMats_Parameters.tCtrlCycleTime := GlobalVariables.tCtrlCycleTime_MAIN;
Controller_OuterCapillaryTubeMats_Parameters.tTaskCycleTime := GlobalVariables.tTaskCycleTime_MAIN;

Controller_OuterCapillaryTubeMats_Permission_Parameters.fHysteresisRange := 6;
Controller_OuterCapillaryTubeMats_Permission_Parameters.tCtrlCycleTime := GlobalVariables.tCtrlCycleTime_MAIN;
Controller_OuterCapillaryTubeMats_Permission_Parameters.tTaskCycleTime := GlobalVariables.tTaskCycleTime_MAIN;


//control strategy for cooling network - fSetpointValue and fActualValue are changed for cooling applications
Controller_OuterCapillaryTubeMats(fSetpointValue := hnltState.fMidTemperature,
	fActualValue := fTargetTemperature_HNLT_Cooling+fOffset_TargetTemperature_OuterCapillaryTubeMats_Cooling,
	eMode := eCTRL_MODE_ACTIVE,
	stParams := Controller_OuterCapillaryTubeMats_Parameters);

//permission controller to ensure that network ist not heated up if ambient temperature is too high
Controller_OuterCapillaryTubeMats_Permission(fSetpointValue := fTargetTemperature_HNLT_Cooling-fOffset_OuterCapillaryTubeMats_Permission,
	fActualValue := ambientState.fOutsideTemperature,
	eMode := eCTRL_MODE_ACTIVE,
	stParams := Controller_OuterCapillaryTubeMats_Permission_Parameters);

hnltControl.bSetStatusOn_OuterCapillaryTubeMats := Controller_OuterCapillaryTubeMats.bOut AND Controller_OuterCapillaryTubeMats_Permission.bOut;	

// turn storages off
hnltControl.bSetStatusOn_HVFASystem := FALSE;
hnltControl.bLoading_HVFASystem := FALSE;
END_METHOD

METHOD ControlHnltCnLinkage : BOOL
VAR_INPUT
END_VAR
//set hysteresis parameters for hnlt cn linkage systems
fOffset_TargetTemperature_HeatPump := 0;
Controller_HeatPump_Parameters.fHysteresisRange := 4;
Controller_HeatPump_Parameters.tCtrlCycleTime := GlobalVariables.tCtrlCycleTime_MAIN;
Controller_HeatPump_Parameters.tTaskCycleTime := GlobalVariables.tTaskCycleTime_MAIN;

fOffset_TargetTemperature_HeatPump_Permission := 3;
Controller_HeatPump_Permission_Parameters.fHysteresisRange := 4;
Controller_HeatPump_Permission_Parameters.tCtrlCycleTime := GlobalVariables.tCtrlCycleTime_MAIN;
Controller_HeatPump_Permission_Parameters.tTaskCycleTime := GlobalVariables.tTaskCycleTime_MAIN;
	
//control heat pump depending on heating demand in hnlt

Controller_HeatPump(fSetpointValue := fTargetTemperature_HNLT_Heating+fOffset_TargetTemperature_HeatPump,
	fActualValue := hnltState.fMidTemperature,
	eMode := eCTRL_MODE_ACTIVE,
	stParams := Controller_HeatPump_Parameters);

Controller_HeatPump_Permission(fSetpointValue := cnState.fMidTemperature,
	fActualValue := fTargetTemperature_CN-fOffset_TargetTemperature_HeatPump_Permission,
	eMode := eCTRL_MODE_ACTIVE,
	stParams := Controller_HeatPump_Parameters);
hnltCnLinkageControl.bSetStatusOn_HeatPump := Controller_HeatPump.bOut AND Controller_HeatPump_Permission.bOut;
hnltCnLinkageControl.fTargetTemperature_ProductionHall := localDefaultParameters.fTargetTemperature_ProductionHall;

hnltCnLinkageControl.bSetStatusOn_InnerCapillaryTubeMats := TRUE;
hnltCnLinkageControl.bSetStatusOn_UnderfloorHeating := TRUE;
END_METHOD

METHOD SetState : BOOL
VAR_INPUT
END_VAR
localState.fTargetTemperature_HNHT_Heating := fTargetTemperature_HNHT_Heating;
localState.fTargetTemperature_HNHT_Cooling := fTargetTemperature_HNHT_Cooling;
localState.fTargetTemperature_HNLT_Heating := fTargetTemperature_HNLT_Heating;
localState.fTargetTemperature_HNLT_Cooling := fTargetTemperature_HNLT_Cooling;
localState.fTargetTemperature_CN := fTargetTemperature_CN;
localState.fTargetTemperature_ProductionHall := localDefaultParameters.fTargetTemperature_ProductionHall;

localState.aTemperatureLimits_HNHT := aTemperatureLimits_HNHT;
localState.aTemperatureLimits_HNLT := aTemperatureLimits_HNLT;
localState.aTemperatureLimits_CN := aTemperatureLimits_CN;	

localState.fFeedTemperature_HNHT := fTargetTemperature_HNHT_Heating+localDefaultParameters.fOffset_FeedTemperature_HNHT;
localState.fFeedTemperature_HNLT_Heating := fTargetTemperature_HNLT_Heating+localDefaultParameters.fOffset_FeedTemperature_HNLT_Heating;
localState.fFeedTemperature_HNLT_Cooling := fTargetTemperature_HNLT_Cooling-localDefaultParameters.fOffset_FeedTemperature_HNLT_Cooling;
localState.fFeedTemperature_CN := fTargetTemperature_CN-localDefaultParameters.fOffset_FeedTemperature_CN;
END_METHOD

METHOD SetTemperatures : BOOL
VAR_INPUT
END_VAR
//set internal variables depending on prodution mode
IF localSetParameters.bProductionModeActivated THEN
	fTargetTemperature_CN := localDefaultParameters.fTargetTemperature_CN_ProductionMode_Summer;
	fTargetTemperature_HNLT_Heating := localDefaultParameters.fTargetTemperature_HNLT_Heating_ProductionMode;
	fTargetTemperature_HNLT_Cooling := localDefaultParameters.fTargetTemperature_HNLT_Cooling_ProductionMode;
	fTargetTemperature_HNHT_Heating := localDefaultParameters.fTargetTemperature_HNHT_Heating_ProductionMode;
	fTargetTemperature_HNHT_Cooling := localDefaultParameters.fTargetTemperature_HNHT_Cooling_ProductionMode;
	aTemperatureLimits_CN := localDefaultParameters.aTemperatureLimits_CN_ProductionMode;
	aTemperatureLimits_HNLT := localDefaultParameters.aTemperatureLimits_HNLT_ProductionMode;
	aTemperatureLimits_HNHT := localDefaultParameters.aTemperatureLimits_HNHT_ProductionMode;

ELSE
	fTargetTemperature_CN := localDefaultParameters.fTargetTemperature_CN_Summer;
	fTargetTemperature_HNLT_Heating := localDefaultParameters.fTargetTemperature_HNLT_Heating;
	fTargetTemperature_HNLT_Cooling := localDefaultParameters.fTargetTemperature_HNLT_Cooling;
	fTargetTemperature_HNHT_Heating := localDefaultParameters.fTargetTemperature_HNHT_Heating;
	fTargetTemperature_HNHT_Cooling := localDefaultParameters.fTargetTemperature_HNHT_Cooling;
	aTemperatureLimits_CN := localDefaultParameters.aTemperatureLimits_CN;
	aTemperatureLimits_HNLT := localDefaultParameters.aTemperatureLimits_HNLT;
	aTemperatureLimits_HNHT := localDefaultParameters.aTemperatureLimits_HNHT;
END_IF

//set feed temperatures
hnhtControl.fFeedTemperature := fTargetTemperature_HNHT_Heating+localDefaultParameters.fOffset_FeedTemperature_HNHT;
hnltControl.fFeedTemperature_Heating := fTargetTemperature_HNLT_Heating+localDefaultParameters.fOffset_FeedTemperature_HNLT_Heating;
hnltControl.fFeedTemperature_Cooling := fTargetTemperature_HNLT_Cooling-localDefaultParameters.fOffset_FeedTemperature_HNLT_Cooling;
cnControl.fFeedTemperature := fTargetTemperature_CN-localDefaultParameters.fOffset_FeedTemperature_CN;
hnhtHnltLinkageControl.fFeedTemperature_HNHT := hnhtControl.fFeedTemperature;
hnhtHnltLinkageControl.fFeedTemperature_HNLT_Heating := hnltControl.fFeedTemperature_Heating;
hnhtHnltLinkageControl.fFeedTemperature_HNLT_Cooling := hnltControl.fFeedTemperature_Cooling;
hnltCnLinkageControl.fFeedTemperature_CN := cnControl.fFeedTemperature;
hnltCnLinkageControl.fFeedTemperature_HNLT_Heating := hnltControl.fFeedTemperature_Heating;
hnltCnLinkageControl.fFeedTemperature_HNLT_Cooling := hnltControl.fFeedTemperature_Cooling;

//set algorithm permission depending on production mode to control structs
CN_Check(fInput := cnState.fMidTemperature,
	fLowerLimit := aTemperatureLimits_CN[1],
	fUpperLimit := aTemperatureLimits_CN[2]);
cnControl.bAlgorithmPermission := CN_Check.bPermission;
	
HNLT_Check(fInput := hnltState.fMidTemperature,
	fLowerLimit := aTemperatureLimits_HNLT[1],
	fUpperLimit := aTemperatureLimits_HNLT[2]);
hnltControl.bAlgorithmPermission := HNLT_Check.bPermission;
	
HNHT_Check(fInput := hnhtState.fMidTemperature,
	fLowerLimit := aTemperatureLimits_HNHT[1],
	fUpperLimit := aTemperatureLimits_HNHT[2]);	
hnhtControl.bAlgorithmPermission := HNHT_Check.bPermission;
	
hnltCnLinkageControl.bAlgorithmPermission_CN := cnControl.bAlgorithmPermission;
hnltCnLinkageControl.bAlgorithmPermission_HNLT := hnltControl.bAlgorithmPermission;
hnhtHnltLinkageControl.bAlgorithmPermission_HNHT := hnhtControl.bAlgorithmPermission;
hnhtHnltLinkageControl.bAlgorithmPermission_HNLT := hnltControl.bAlgorithmPermission;
hnhtCnLinkageControl.bAlgorithmPermission_CN := cnControl.bAlgorithmPermission;
hnhtCnLinkageControl.bAlgorithmPermission_HNHT := hnhtControl.bAlgorithmPermission;
END_METHOD

END_FUNCTION_BLOCK

// ---- POUs/06 Strategy/FB_StrategyController_Conventional.TcPOU
FUNCTION_BLOCK FB_StrategyController_Conventional
VAR_INPUT
	ambientState : ST_AmbientState;
	
	//actual temperatures in thermal networks
	cnState : ST_ThermalNetworkState;
	hnltState : ST_ThermalNetworkState;
	hnhtState : ST_ThermalNetworkState;
END_VAR
VAR_OUTPUT	
	cnControl : ST_CoolingNetworkControl;
	hnltControl : ST_HeatingNetworkLowTemperatureControl;	
	hnhtControl : ST_HeatingNetworkHighTemperatureControl;
	hnltCnLinkageControl : ST_HnltCnLinkageControl;
	hnhtHnltLinkageControl : ST_HnhtHnltLinkageControl;
	hnhtCnLinkageControl : ST_HnhtCnLinkageControl;
END_VAR
VAR
	{attribute 'OPC.UA.DA' := '1'}
	localSetParameters : ST_StrategySetParameters;	
	{attribute 'OPC.UA.DA' := '1'}
	localState : ST_StrategyState;	

	//default parameters
	localDefaultParameters : ST_StrategyDefaultParameters;

	//internal variables
	fTargetTemperature_HNHT_Heating : REAL;
	fTargetTemperature_HNHT_Cooling : REAL;
	fTargetTemperature_HNLT_Cooling : REAL;
	fTargetTemperature_HNLT_Heating : REAL;
	fTargetTemperature_CN : REAL;
	aTemperatureLimits_HNHT : ARRAY[1..2] OF REAL;
	aTemperatureLimits_HNLT : ARRAY[1..2] OF REAL;
	aTemperatureLimits_CN : ARRAY[1..2] OF REAL;
	stHNHTCheckDefaultParameters : ST_RangeCheckDefaultParameters := (tTaskCycleTime := GlobalVariables.tCtrlCycleTime_MAIN, tCtrlCycleTime := GlobalVariables.tCtrlCycleTime_MAIN, fRestoreDifference := 5);
	HNHT_Check : FB_RangeCheck := (ST_DefaultParameters := stHNHTCheckDefaultParameters);
	stHNLTCheckDefaultParameters : ST_RangeCheckDefaultParameters := (tTaskCycleTime := GlobalVariables.tCtrlCycleTime_MAIN, tCtrlCycleTime := GlobalVariables.tCtrlCycleTime_MAIN, fRestoreDifference := 5);
	HNLT_Check : FB_RangeCheck := (ST_DefaultParameters := stHNLTCheckDefaultParameters);
	stCNCheckDefaultParameters : ST_RangeCheckDefaultParameters := (tTaskCycleTime := GlobalVariables.tCtrlCycleTime_MAIN, tCtrlCycleTime := GlobalVariables.tCtrlCycleTime_MAIN, fRestoreDifference := 2);
	CN_Check : FB_RangeCheck := (ST_DefaultParameters := stCNCheckDefaultParameters);
	
	//controller and variables for high temperature heating network

	Controller_CondensingBoiler : FB_CTRL_2POINT;
	Controller_CondensingBoiler_Parameters : ST_CTRL_2POINT_PARAMS;
	Controller_StaticHeating : FB_CTRL_2POINT;
	Controller_StaticHeating_Parameters : ST_CTRL_2POINT_PARAMS;
	
	//controllers and variables for low temperature heating network
	Controller_OuterCapillaryTubeMats : FB_CTRL_2POINT;
	Controller_OuterCapillaryTubeMats_Parameters : ST_CTRL_2POINT_PARAMS;
	Controller_OuterCapillaryTubeMats_Permission : FB_CTRL_2POINT;
	Controller_OuterCapillaryTubeMats_Permission_Parameters : ST_CTRL_2POINT_PARAMS;
	fOffset_TargetTemperature_OuterCapillaryTubeMats_Cooling : REAL := 1;	
	fOffset_OuterCapillaryTubeMats_Permission : REAL := 10;
	
	//controllers and variables for cooling network
	fOffset_TargetTemperature_eChiller : REAL := 0.5;	
	Controller_eChiller : FB_CTRL_2POINT;
	Controller_eChiller_Parameters : ST_CTRL_2POINT_PARAMS;	

	//controllers and variables for hnht and hnlt linkage
	Controller_HeatExchanger1_HNHT : FB_CTRL_2POINT;
	Controller_HeatExchanger1_HNHT_Parameters : ST_CTRL_2POINT_PARAMS;	
	Controller_HeatExchanger1_HNLT : FB_CTRL_2POINT;
	Controller_HeatExchanger1_HNLT_Parameters : ST_CTRL_2POINT_PARAMS;
	fOffset_TargetTemperature_HeatExchanger1 : REAL := 2;

	//clock
	stDefaultParameters_Clock : ST_ClockDefaultParameters := (tTaskCycleTime := GlobalVariables.tCtrlCycleTime_MAIN, tCtrlCycleTime := T#1M);
	Clock : FB_Clock := (ST_DefaultParameters := stDefaultParameters_Clock);
END_VAR

Clock();
AmbientControl();
SetTemperatures();
ControlCN();
ControlHNLT();
ControlHNHT();
ControlHnltCnLinkage();
ControlHnhtHnltLinkage();
SetState();

METHOD AmbientControl : BOOL
VAR_INPUT
END_VAR
//check for heating or cooling mode
IF Clock.stClockState.sintMonth>4 AND Clock.stClockState.sintMonth<10 THEN
	//heating mode
	hnltCnLinkageControl.bHeatingMode := FALSE;
	hnhtCnLinkageControl.bHeatingMode := FALSE;
ELSE
	//cooling mode	
	hnltCnLinkageControl.bHeatingMode := TRUE;
	hnhtCnLinkageControl.bHeatingMode := TRUE;
END_IF
END_METHOD

METHOD ControlCN : BOOL
VAR_INPUT
END_VAR
//set hysteresis parameters for two-point controllers in cooling network
Controller_eChiller_Parameters.fHysteresisRange := 7;
Controller_eChiller_Parameters.tCtrlCycleTime := GlobalVariables.tCtrlCycleTime_MAIN;
Controller_eChiller_Parameters.tTaskCycleTime := GlobalVariables.tTaskCycleTime_MAIN;

//control eChiller
Controller_eChiller(fSetpointValue := cnState.fMidTemperature,
	fActualValue := fTargetTemperature_CN-fOffset_TargetTemperature_eChiller,
	eMode := eCTRL_MODE_ACTIVE,
	stParams := Controller_eChiller_Parameters);

cnControl.bSetStatusOn_eChiller := Controller_eChiller.bOut;

//set HFVA off
cnControl.bSetStatusOn_HVFASystem := FALSE;
cnControl.bLoading_HVFASystem := FALSE;
END_METHOD

METHOD ControlHNHT : BOOL
VAR_INPUT
END_VAR
VAR
END_VAR
Controller_CondensingBoiler_Parameters.fHysteresisRange := 12;
Controller_CondensingBoiler_Parameters.tCtrlCycleTime := GlobalVariables.tCtrlCycleTime_MAIN;
Controller_CondensingBoiler_Parameters.tTaskCycleTime := GlobalVariables.tTaskCycleTime_MAIN;

Controller_StaticHeating_Parameters.fHysteresisRange := 4;
Controller_StaticHeating_Parameters.tCtrlCycleTime := GlobalVariables.tCtrlCycleTime_MAIN;
Controller_StaticHeating_Parameters.tTaskCycleTime := GlobalVariables.tTaskCycleTime_MAIN;


IF (Clock.stClockState.sintWeekday > 0 AND Clock.stClockState.sintWeekday < 6) AND (Clock.stClockState.fHour > 5 AND Clock.stClockState.fHour < 23) THEN
	hnhtControl.bSetStatusOn_CHP1 := TRUE;
	hnhtControl.bSetStatusOn_CHP2 := TRUE;
ELSE
	hnhtControl.bSetStatusOn_CHP1 := FALSE;
	hnhtControl.bSetStatusOn_CHP2 := FALSE;
END_IF

//condensing boiler is switched if network temperature falls below critical temperature limit
Controller_CondensingBoiler(fSetpointValue := fTargetTemperature_HNHT_Heating,
	fActualValue := hnhtState.fUpperTemperature,
	eMode := eCTRL_MODE_ACTIVE,
	stParams := Controller_CondensingBoiler_Parameters);
hnhtControl.bSetStatusOn_CondensingBoiler := Controller_CondensingBoiler.bOut;


hnhtControl.bSetStatusOn_VSIStorage := FALSE;
hnhtControl.bLoading_VSISystem := FALSE;


Controller_StaticHeating(fSetpointValue := 15,
	fActualValue := ambientState.fOutsideTemperature,
	eMode := eCTRL_MODE_ACTIVE,
	stParams := Controller_StaticHeating_Parameters);
hnhtControl.bSetStatusOn_StaticHeating := Controller_StaticHeating.bOut;
END_METHOD

METHOD ControlHnhtHnltLinkage : BOOL
VAR_INPUT
END_VAR
Controller_HeatExchanger1_HNHT_Parameters.fHysteresisRange := 8;
Controller_HeatExchanger1_HNHT_Parameters.tCtrlCycleTime := GlobalVariables.tCtrlCycleTime_MAIN;
Controller_HeatExchanger1_HNHT_Parameters.tTaskCycleTime := GlobalVariables.tTaskCycleTime_MAIN;

Controller_HeatExchanger1_HNLT_Parameters.fHysteresisRange := 8;
Controller_HeatExchanger1_HNLT_Parameters.tCtrlCycleTime := GlobalVariables.tCtrlCycleTime_MAIN;
Controller_HeatExchanger1_HNLT_Parameters.tTaskCycleTime := GlobalVariables.tTaskCycleTime_MAIN;


//control heat exchanger 1 from HNHT
Controller_HeatExchanger1_HNHT(fSetpointValue := hnhtState.fUpperTemperature,
	fActualValue := fTargetTemperature_HNHT_Cooling,
	eMode := eCTRL_MODE_ACTIVE,
	stParams := Controller_HeatExchanger1_HNHT_Parameters);

//control heat exchanger 1 from HNLT
Controller_HeatExchanger1_HNLT(fSetpointValue := fTargetTemperature_HNLT_Heating-fOffset_TargetTemperature_HeatExchanger1,
	fActualValue := hnltState.fMidTemperature,
	eMode := eCTRL_MODE_ACTIVE,
	stParams := Controller_HeatExchanger1_HNLT_Parameters);
	
hnhtHnltLinkageControl.bSetStatusOn_HeatExchanger1 := Controller_HeatExchanger1_HNHT.bOut OR Controller_HeatExchanger1_HNLT.bOut;

//turn heat pump off
hnhtHnltLinkageControl.bSetStatusOn_HeatPump := FALSE;
END_METHOD

METHOD ControlHNLT : BOOL
VAR_INPUT
END_VAR
//set hysteresis parameters for two-point controllers in cooling network
Controller_OuterCapillaryTubeMats_Parameters.fHysteresisRange := 6;
Controller_OuterCapillaryTubeMats_Parameters.tCtrlCycleTime := GlobalVariables.tCtrlCycleTime_MAIN;
Controller_OuterCapillaryTubeMats_Parameters.tTaskCycleTime := GlobalVariables.tTaskCycleTime_MAIN;

Controller_OuterCapillaryTubeMats_Permission_Parameters.fHysteresisRange := 6;
Controller_OuterCapillaryTubeMats_Permission_Parameters.tCtrlCycleTime := GlobalVariables.tCtrlCycleTime_MAIN;
Controller_OuterCapillaryTubeMats_Permission_Parameters.tTaskCycleTime := GlobalVariables.tTaskCycleTime_MAIN;


//control strategy for cooling network - fSetpointValue and fActualValue are changed for cooling applications
Controller_OuterCapillaryTubeMats(fSetpointValue := hnltState.fMidTemperature,
	fActualValue := fTargetTemperature_HNLT_Cooling+fOffset_TargetTemperature_OuterCapillaryTubeMats_Cooling,
	eMode := eCTRL_MODE_ACTIVE,
	stParams := Controller_OuterCapillaryTubeMats_Parameters);

//permission controller to ensure that network ist not heated up if ambient temperature is too high
Controller_OuterCapillaryTubeMats_Permission(fSetpointValue := fTargetTemperature_HNLT_Cooling-fOffset_OuterCapillaryTubeMats_Permission,
	fActualValue := ambientState.fOutsideTemperature,
	eMode := eCTRL_MODE_ACTIVE,
	stParams := Controller_OuterCapillaryTubeMats_Permission_Parameters);

hnltControl.bSetStatusOn_OuterCapillaryTubeMats := Controller_OuterCapillaryTubeMats.bOut AND Controller_OuterCapillaryTubeMats_Permission.bOut;

// turn HFVA off
hnltControl.bSetStatusOn_HVFASystem := FALSE;
hnltControl.bLoading_HVFASystem := FALSE;
END_METHOD

METHOD ControlHnltCnLinkage : BOOL
VAR_INPUT
END_VAR

// set heat pump off
hnltCnLinkageControl.bSetStatusOn_HeatPump := FALSE;


hnltCnLinkageControl.fTargetTemperature_ProductionHall := localDefaultParameters.fTargetTemperature_ProductionHall;

hnltCnLinkageControl.bSetStatusOn_InnerCapillaryTubeMats := TRUE;
hnltCnLinkageControl.bSetStatusOn_UnderfloorHeating := TRUE;
END_METHOD

METHOD SetState : BOOL
VAR_INPUT
END_VAR
localState.fTargetTemperature_HNHT_Heating := fTargetTemperature_HNHT_Heating;
localState.fTargetTemperature_HNHT_Cooling := fTargetTemperature_HNHT_Cooling;
localState.fTargetTemperature_HNLT_Heating := fTargetTemperature_HNLT_Heating;
localState.fTargetTemperature_HNLT_Cooling := fTargetTemperature_HNLT_Cooling;
localState.fTargetTemperature_CN := fTargetTemperature_CN;
localState.fTargetTemperature_ProductionHall := localDefaultParameters.fTargetTemperature_ProductionHall;

localState.aTemperatureLimits_HNHT := aTemperatureLimits_HNHT;
localState.aTemperatureLimits_HNLT := aTemperatureLimits_HNLT;
localState.aTemperatureLimits_CN := aTemperatureLimits_CN;	

localState.fFeedTemperature_HNHT := fTargetTemperature_HNHT_Heating+localDefaultParameters.fOffset_FeedTemperature_HNHT;
localState.fFeedTemperature_HNLT_Heating := fTargetTemperature_HNLT_Heating+localDefaultParameters.fOffset_FeedTemperature_HNLT_Heating;
localState.fFeedTemperature_HNLT_Cooling := fTargetTemperature_HNLT_Cooling-localDefaultParameters.fOffset_FeedTemperature_HNLT_Cooling;
localState.fFeedTemperature_CN := fTargetTemperature_CN-localDefaultParameters.fOffset_FeedTemperature_CN;
END_METHOD

METHOD SetTemperatures : BOOL
VAR_INPUT
END_VAR
//set internal variables depending on prodution mode
IF localSetParameters.bProductionModeActivated THEN
	fTargetTemperature_CN := localDefaultParameters.fTargetTemperature_CN_ProductionMode_Summer;	
	fTargetTemperature_HNLT_Heating := localDefaultParameters.fTargetTemperature_HNLT_Heating_ProductionMode;
	fTargetTemperature_HNLT_Cooling := localDefaultParameters.fTargetTemperature_HNLT_Cooling_ProductionMode;
	fTargetTemperature_HNHT_Heating := localDefaultParameters.fTargetTemperature_HNHT_Heating_ProductionMode;
	fTargetTemperature_HNHT_Cooling := localDefaultParameters.fTargetTemperature_HNHT_Cooling_ProductionMode;
	aTemperatureLimits_CN := localDefaultParameters.aTemperatureLimits_CN_ProductionMode;
	aTemperatureLimits_HNLT := localDefaultParameters.aTemperatureLimits_HNLT_ProductionMode;
	aTemperatureLimits_HNHT := localDefaultParameters.aTemperatureLimits_HNHT_ProductionMode;

ELSE
	fTargetTemperature_CN := localDefaultParameters.fTargetTemperature_CN_Summer;
	fTargetTemperature_HNLT_Heating := localDefaultParameters.fTargetTemperature_HNLT_Heating;
	fTargetTemperature_HNLT_Cooling := localDefaultParameters.fTargetTemperature_HNLT_Cooling;
	fTargetTemperature_HNHT_Heating := localDefaultParameters.fTargetTemperature_HNHT_Heating;
	fTargetTemperature_HNHT_Cooling := localDefaultParameters.fTargetTemperature_HNHT_Cooling;
	aTemperatureLimits_CN := localDefaultParameters.aTemperatureLimits_CN;
	aTemperatureLimits_HNLT := localDefaultParameters.aTemperatureLimits_HNLT;
	aTemperatureLimits_HNHT := localDefaultParameters.aTemperatureLimits_HNHT;
END_IF

